// TIA Portal project "V1.3" (V16)

(* hardware
DEVICE "S7-1200 station_1"  S7-1200 Station
   slot 0: "Rack_0"  S7-1200 Rack  Rack  V1.0
   slot 1: "PLC_1"  CPU 1214C DC/DC/DC  6ES7 214-1AG40-0XB0  V4.2
   slot 2: "DI 16/DQ 16x24VDC_1"  6ES7 223-1BL32-0XB0  V2.0
   slot 3: "DI 16x24VDC/DQ 16xRelay_1"  SM 1223 DI16/DQ16 x relay  6ES7 223-1PL32-0XB0  V2.0
   slot 3: "AI 1x12BIT_1"  AI1 signal board  6ES7 231-4HA30-0XB0  V2.0
DEVICE "HMI_1"  KTP700 Basic PN
   slot 0: "HMI_1"  KTP700 Basic PN  6AV2 123-2GB03-0AX0  15.0.0.0
   slot 1: "HMI_RT_1"  KTP700 Basic PN  6AV2 123-2GB03-0AX0  15.0.0.0
   slot 5: "HMI_1.IE_CP_1"  PROFINET Interface  15.0.0.0
      slot 1: "PROFINET Interface_1"  PROFINET Interface
         slot 1: "Port_1"  Port
*)

// ===== PLC "PLC_1"  CPU 1214C DC/DC/DC =====

VAR_GLOBAL   // PLC tag table "Default tag table"
   "czujnik ciśnienia powietrza" AT %I0.0 : Bool;
   "ESTOP" AT %I0.1 : Bool;
   "[P] załączenie powietrza" AT %I0.2 : Bool;
   "[P] wyłączenie powietrza [NC]" AT %I0.3 : Bool;
   "[P] załączenie pompy hydraulicznej" AT %I0.4 : Bool;
   "[P] wyłączenie pompy hydraulicznej [NC]" AT %I0.5 : Bool;
   "[P] przycisk dwuręczny [NC]" AT %I0.6 : Bool;
   "[P] przycisk dwuręczny [NO]" AT %I0.7 : Bool;
   "SQ1" AT %I1.0 : Bool;
   "SQ2" AT %I1.1 : Bool;
   "SQ3" AT %I1.2 : Bool;
   "SQ4" AT %I1.3 : Bool;
   "SQ5" AT %I1.4 : Bool;
   "SQ6" AT %I1.5 : Bool;
   "Bit_1" AT %I8.0 : Bool;
   "Bit_2" AT %I8.1 : Bool;
   "Bit_3" AT %I8.2 : Bool;
   "Bit_4" AT %I8.3 : Bool;
   "Bit_5" AT %I8.4 : Bool;
   "Bit_6" AT %I8.5 : Bool;
   "zwierny_1" AT %I8.6 : Bool;
   "zwierny_2" AT %I8.7 : Bool;
   "zwierny_3" AT %I9.0 : Bool;
   "zwierny_4" AT %I9.1 : Bool;
   "zwierny_5" AT %I9.2 : Bool;
   "zwierny_6" AT %I9.3 : Bool;
   "-" AT %I9.4 : Bool;
   "-(1)" AT %I9.5 : Bool;
   "-(2)" AT %I9.6 : Bool;
   "-(3)" AT %I9.7 : Bool;
   "-(4)" AT %I12.0 : Bool;
   "-(5)" AT %I12.1 : Bool;
   "-(6)" AT %I12.2 : Bool;
   "-(7)" AT %I12.3 : Bool;
   "-(8)" AT %I12.4 : Bool;
   "-(9)" AT %I12.5 : Bool;
   "-(10)" AT %I12.6 : Bool;
   "Kurtyna" AT %I12.7 : Bool;
   "-(12)" AT %I13.0 : Bool;
   "-(13)" AT %I13.1 : Bool;
   "-(14)" AT %I13.2 : Bool;
   "-(15)" AT %I13.3 : Bool;
   "-(16)" AT %I13.4 : Bool;
   "-(17)" AT %I13.5 : Bool;
   "-(18)" AT %I13.6 : Bool;
   "-(19)" AT %I13.7 : Bool;
   "Ciśnienie oleju hydraulicznego" AT %IW80 : Int;
   "Z.H 0" AT %Q0.0 : Bool;
   "Z.H 1" AT %Q0.1 : Bool;
   "Z.H 2" AT %Q0.2 : Bool;
   "Z.H 3" AT %Q0.3 : Bool;
   "Z.H 4" AT %Q0.4 : Bool;
   "Z.H 5" AT %Q0.5 : Bool;
   "Z.H 6" AT %Q0.6 : Bool;
   "Z.H 7" AT %Q0.7 : Bool;
   "Z.H 8" AT %Q1.0 : Bool;
   "-(20)" AT %Q1.1 : Bool;
   "[L] Zawór główny powietrza" AT %Q8.0 : Bool;
   "[L] Pompa hydrauliczna" AT %Q8.1 : Bool;
   "-(21)" AT %Q8.2 : Bool;
   "-(22)" AT %Q8.3 : Bool;
   "-(23)" AT %Q8.4 : Bool;
   "-(24)" AT %Q8.5 : Bool;
   "-(25)" AT %Q8.6 : Bool;
   "-(26)" AT %Q8.7 : Bool;
   "Proces1" AT %Q9.0 : Bool;
   "Proces2" AT %Q9.1 : Bool;
   "Proces3" AT %Q9.2 : Bool;
   "Proces4" AT %Q9.3 : Bool;
   "Proces5" AT %Q9.4 : Bool;
   "Proces6" AT %Q9.5 : Bool;
   "Proces7" AT %Q9.6 : Bool;
   "Proces8" AT %Q9.7 : Bool;
   "Z.P 0" AT %Q12.0 : Bool;
   "Z.P 1" AT %Q12.1 : Bool;
   "Z.P 2" AT %Q12.2 : Bool;
   "Z.P 3" AT %Q12.3 : Bool;
   "Z.P 4" AT %Q12.4 : Bool;
   "smar 1" AT %Q12.5 : Bool;
   "smar 2" AT %Q12.6 : Bool;
   "-(27)" AT %Q12.7 : Bool;
   "-(28)" AT %Q13.0 : Bool;
   "-(29)" AT %Q13.1 : Bool;
   "-(30)" AT %Q13.2 : Bool;
   "-(31)" AT %Q13.3 : Bool;
   "Pompa hydrauliczna" AT %Q13.4 : Bool;
   "-(33)" AT %Q13.5 : Bool;
   "-(34)" AT %Q13.6 : Bool;
   "-(35)" AT %Q13.7 : Bool;
   "Bit1(1)" AT %M0.0 : Bool;
   "Bit2(1)" AT %M0.1 : Bool;
   "Bit3(1)" AT %M0.2 : Bool;
   "Bit4(1)" AT %M0.3 : Bool;
   "Bit5(1)" AT %M0.4 : Bool;
   "Bit6(1)" AT %M0.5 : Bool;
   "Byte0" AT %MB0 : Byte;
   "Tag_1" AT %M7000.0 : Bool;
   "Tag_2" AT %M7000.1 : Bool;
   "Tag_3" AT %M7000.2 : Bool;
   "Tag_4" AT %M7000.5 : Bool;
END_VAR

DATA_BLOCK "main_DB"   // DB2
{ S7_Optimized_Access := 'TRUE' }
VERSION : 0.1
   VAR
      "M" : Array[0..254] of Bool;
      Button : Struct
         Screen_0 : Struct
            Reset_counter_1 : Bool;
            Reset_counter_2 : Bool;
            Lubrication_test : Bool;
            Lubrication_test_1 : Bool;
            Lubrication_test_2 : Bool;
         END_STRUCT;
         Screen_2 : Struct
            "Z.P 0" : Bool;
            "Z.P 1" : Bool;
            "Z.P 2" : Bool;
            "Z.P 3" : Bool;
            "Z.P 4" : Bool;
            "Z.H 0" : Bool;
            "Z.H 1" : Bool;
            "Z.H 2" : Bool;
            "Z.H 3" : Bool;
            "Z.H 4" : Bool;
            "Z.H 5" : Bool;
            "Z.H 6" : Bool;
            "Z.H 7" : Bool;
            "Z.H 8" : Bool;
            Manual_control : Bool;
            Hydraulic_Pump : Bool;
            Relaxation : Bool;
         END_STRUCT;
         Screen_1 : Struct
            "0" : Bool;
         END_STRUCT;
         Screen_3 : Struct
            "0" : Bool;
         END_STRUCT;
         Template : Struct
            "Browsed_punch_+" : Bool;
            "Browsed_punch_-" : Bool;
         END_STRUCT;
      END_STRUCT;
      Status : Struct
         Blink : Bool;
         Manual_control : Bool;
         Browsing_punch : Bool;
         "Two-handed_button" : Bool;
         relaxation : Bool;
         Cycle_time_overload : Bool;
         Lubrication1 : Bool;
         Lubrication2 : Bool;
      END_STRUCT;
   END_VAR
   VAR RETAIN
      var : Struct
         Browsed_punch : Byte;
         Connected_punch : Byte;
         Result_punch : Byte;
         Hydraulic_oil_pressure : Real;
         Lubrication_dur : Time;
         Lubrication_frequency : Int := 1;
         "Descryption Z.P 1" : String;
         "Descryption Z.P 2" : String;
         "Descryption Z.P 3" : String;
         "Descryption Z.P 4" : String;
         "Descryption Z.H 1" : String;
         "Descryption Z.H 2" : String;
         "Descryption Z.H 3" : String;
         "Descryption Z.H 4" : String;
         "Descryption Z.H 5" : String;
         "Descryption Z.H 6" : String;
         "Descryption Z.H 7" : String;
         "Descryption Z.H 8" : String;
         "Descryption SQ 1" : String;
         "Descryption SQ 2" : String;
         "Descryption SQ 3" : String;
         "Descryption SQ 4" : String;
         "Descryption SQ 5" : String;
         "Descryption SQ 6" : String;
         "Descryption contact_sensor 1" : String;
         "Descryption contact_sensor 2" : String;
         "Descryption contact_sensor 3" : String;
         "Descryption contact_sensor 4" : String;
         "Descryption contact_sensor 5" : String;
         "Descryption contact_sensor 6" : String;
      END_STRUCT;
   END_VAR
   VAR
      Timers : Struct
         "0" : IEC_TIMER;
         "1" : IEC_TIMER;
         "2" : IEC_TIMER;
         "3" : IEC_TIMER;
         "4" : IEC_TIMER;
         "5" : IEC_TIMER;
         "6" : IEC_TIMER;
         "7" : IEC_TIMER;
         "8" : IEC_TIMER;
         "9" : IEC_TIMER;
         "10" : IEC_TIMER;
         "11" : IEC_TIMER;
         "12" : IEC_TIMER;
         "13" : IEC_TIMER;
         "14" : IEC_TIMER;
         "15" : IEC_TIMER;
         "16" : IEC_TIMER;
         "17" : IEC_TIMER;
         "18" : IEC_TIMER;
         "19" : IEC_TIMER;
         "20" : IEC_TIMER;
         "21" : IEC_TIMER;
         "22" : IEC_TIMER;
         "23" : IEC_TIMER;
         "24" : IEC_TIMER;
      END_STRUCT;
   END_VAR
BEGIN
END_DATA_BLOCK

DATA_BLOCK "Counters"   // DB5
{ S7_Optimized_Access := 'TRUE' }
VERSION : 0.1
   VAR RETAIN
      Counter_1 : Int;
      Counter_2 : Int;
   END_VAR
   VAR
      Lubricatons : Int := 1;
   END_VAR
BEGIN
END_DATA_BLOCK

DATA_BLOCK "Punch_parameters"   // DB6
{ S7_Optimized_Access := 'TRUE' }
VERSION : 0.1
   VAR
      Punch : Array[0..10] of Struct
         "Z.P 1" : String;
         "Z.P 2" : String;
         "Z.P 3" : String;
         "Z.P 4" : String;
         "Z.H 1" : String;
         "Z.H 2" : String;
         "Z.H 3" : String;
         "Z.H 4" : String;
         "Z.H 5" : String;
         "Z.H 6" : String;
         "Z.H 7" : String;
         "Z.H 8" : String;
         SQ1 : String;
         SQ2 : String;
         SQ3 : String;
         SQ4 : String;
         SQ5 : String;
         SQ6 : String;
         Contact_sensor_1 : String;
         Contact_sensor_2 : String;
         Contact_sensor_3 : String;
         Contact_sensor_4 : String;
         Contact_sensor_5 : String;
         Contact_sensor_6 : String;
      END_STRUCT;
   END_VAR
BEGIN
   Punch[1]."Z.H 5" := 'Lewy naprzod';
   Punch[1]."Z.H 6" := 'Lewy wstecz';
   Punch[1]."Z.H 7" := 'Prawy naprzod';
   Punch[1]."Z.H 8" := 'Prawy wstecz';
   Punch[1].SQ1 := 'Lewy z tylu [NC]';
   Punch[1].SQ2 := 'Lewy z przodu';
   Punch[1].SQ3 := 'Prawy z tylu';
   Punch[1].SQ4 := 'Prawy z przodu';
   Punch[1].Contact_sensor_1 := 'Przy lewym silowniku';
   Punch[1].Contact_sensor_2 := 'Przy prawym silowniku 1';
   Punch[1].Contact_sensor_3 := 'Przy prawym silowniku 2';
   Punch[1]."Z.P 1" := 'Klamra';
   Punch[1]."Z.P 2" := 'Baza';
   Punch[1].SQ5 := 'Klamra zacisnieta';
   Punch[2]."Z.P 1" := 'Baza';
   Punch[2]."Z.P 2" := 'Kon';
   Punch[2].SQ3 := 'Kon';
   Punch[2]."Z.H 1" := 'Silownik naprzod';
   Punch[2]."Z.H 2" := 'Silownik wstecz';
   Punch[2].SQ1 := 'Silownik przod';
   Punch[2].SQ2 := 'Silownik tyl';
   Punch[2].Contact_sensor_1 := '1';
   Punch[2].Contact_sensor_2 := '2';
   Punch[3]."Z.P 1" := 'Kon 1';
   Punch[3]."Z.P 2" := 'Kon 2';
   Punch[3]."Z.H 3" := 'Silownik naprzod';
   Punch[3]."Z.H 4" := 'Silownik wstecz';
   Punch[3].SQ1 := 'Silownik przod';
   Punch[3].SQ2 := 'Silownik tyl';
   Punch[3].SQ3 := 'Kon 1';
   Punch[3].SQ4 := 'Kon 2';
   Punch[3].Contact_sensor_1 := '1';
   Punch[3].Contact_sensor_2 := '2';
   Punch[4].SQ1 := 'Prawy stempel wysuniety';
   Punch[4].Contact_sensor_1 := '1';
   Punch[4].SQ2 := 'Prawy stempel wycofany';
   Punch[4].SQ3 := 'Lewy stempel wysuniety';
   Punch[4].SQ4 := 'Lewy stempel wycofany';
   Punch[4]."Z.H 1" := 'L st. wysuniecie';
   Punch[4]."Z.H 2" := 'L st. wycofanie';
   Punch[4]."Z.H 3" := 'P st. wysuniecie';
   Punch[4]."Z.H 4" := 'P st. wycofanie';
   Punch[5]."Z.H 7" := 'Stempel naprzod';
   Punch[5]."Z.H 8" := 'Stempel wstecz';
   Punch[5].SQ1 := 'Material dosuniety';
   Punch[5].SQ2 := 'Stempel wycofany';
END_DATA_BLOCK

DATA_BLOCK "Relaxation_DB"   // DB7
{ S7_Optimized_Access := 'TRUE' }
VERSION : 0.1
// stored: InstanceOfName Relaxation
"Relaxation"
BEGIN
END_DATA_BLOCK

// folder: Punch_blocks

DATA_BLOCK "Punch1_DB"   // DB1
{ S7_Optimized_Access := 'TRUE' }
VERSION : 0.1
// stored: InstanceOfName Punch1
"Punch1"
BEGIN
END_DATA_BLOCK

DATA_BLOCK "Punch2_DB"   // DB3
{ S7_Optimized_Access := 'TRUE' }
VERSION : 0.1
// stored: InstanceOfName Punch2
"Punch2"
BEGIN
END_DATA_BLOCK

DATA_BLOCK "Punch3_DB"   // DB4
{ S7_Optimized_Access := 'TRUE' }
VERSION : 0.1
// stored: InstanceOfName Punch3
"Punch3"
BEGIN
END_DATA_BLOCK

DATA_BLOCK "Punch4_DB"   // DB15
{ S7_Optimized_Access := 'TRUE' }
VERSION : 0.1
// stored: InstanceOfName Punch4
"Punch4"
BEGIN
END_DATA_BLOCK

DATA_BLOCK "Punch5_DB"   // DB16
{ S7_Optimized_Access := 'TRUE' }
VERSION : 0.1
// stored: InstanceOfName Punch5
"Punch5"
BEGIN
END_DATA_BLOCK

// folder: System blocks/Program resources

DATA_BLOCK "IEC_Timer_0_DB"   // DB8
{ S7_Optimized_Access := 'TRUE' }
AUTHOR : Simatic
FAMILY : IEC
NAME : IEC_TMR
VERSION : 1.0
// stored: InstanceOfName IEC_TIMER
"IEC_TIMER"
BEGIN
END_DATA_BLOCK

DATA_BLOCK "IEC_Timer_0_DB_1"   // DB9
{ S7_Optimized_Access := 'TRUE' }
AUTHOR : Simatic
FAMILY : IEC
NAME : IEC_TMR
VERSION : 1.0
// stored: InstanceOfName IEC_TIMER
"IEC_TIMER"
BEGIN
END_DATA_BLOCK

DATA_BLOCK "IEC_Timer_0_DB_2"   // DB10
{ S7_Optimized_Access := 'TRUE' }
AUTHOR : Simatic
FAMILY : IEC
NAME : IEC_TMR
VERSION : 1.0
// stored: InstanceOfName IEC_TIMER
"IEC_TIMER"
BEGIN
END_DATA_BLOCK

DATA_BLOCK "IEC_Timer_0_DB_3"   // DB11
{ S7_Optimized_Access := 'TRUE' }
AUTHOR : Simatic
FAMILY : IEC
NAME : IEC_TMR
VERSION : 1.0
// stored: InstanceOfName IEC_TIMER
"IEC_TIMER"
BEGIN
END_DATA_BLOCK

DATA_BLOCK "IEC_Timer_0_DB_4"   // DB12
{ S7_Optimized_Access := 'TRUE' }
AUTHOR : Simatic
FAMILY : IEC
NAME : IEC_TMR
VERSION : 1.0
// stored: InstanceOfName IEC_TIMER
"IEC_TIMER"
BEGIN
END_DATA_BLOCK

DATA_BLOCK "IEC_Timer_0_DB_5"   // DB13
{ S7_Optimized_Access := 'TRUE' }
AUTHOR : Simatic
FAMILY : IEC
NAME : IEC_TMR
VERSION : 1.0
// stored: InstanceOfName IEC_TIMER
"IEC_TIMER"
BEGIN
END_DATA_BLOCK

DATA_BLOCK "IEC_Timer_0_DB_6"   // DB14
{ S7_Optimized_Access := 'TRUE' }
AUTHOR : Simatic
FAMILY : IEC
NAME : IEC_TMR
VERSION : 1.0
// stored: InstanceOfName IEC_TIMER
"IEC_TIMER"
BEGIN
END_DATA_BLOCK

// folder: (top level)

FUNCTION_BLOCK "Relaxation"   // FB4, LAD
{ S7_Optimized_Access := 'TRUE' }
VERSION : 0.1
   VAR_INPUT
      Activate : Bool;
   END_VAR
   VAR
      finish : Bool;
   END_VAR
   VAR_TEMP   // added for the SCL form of the ladder/FBD networks
      _w1 : Bool;
   END_VAR
BEGIN

REGION Network 1
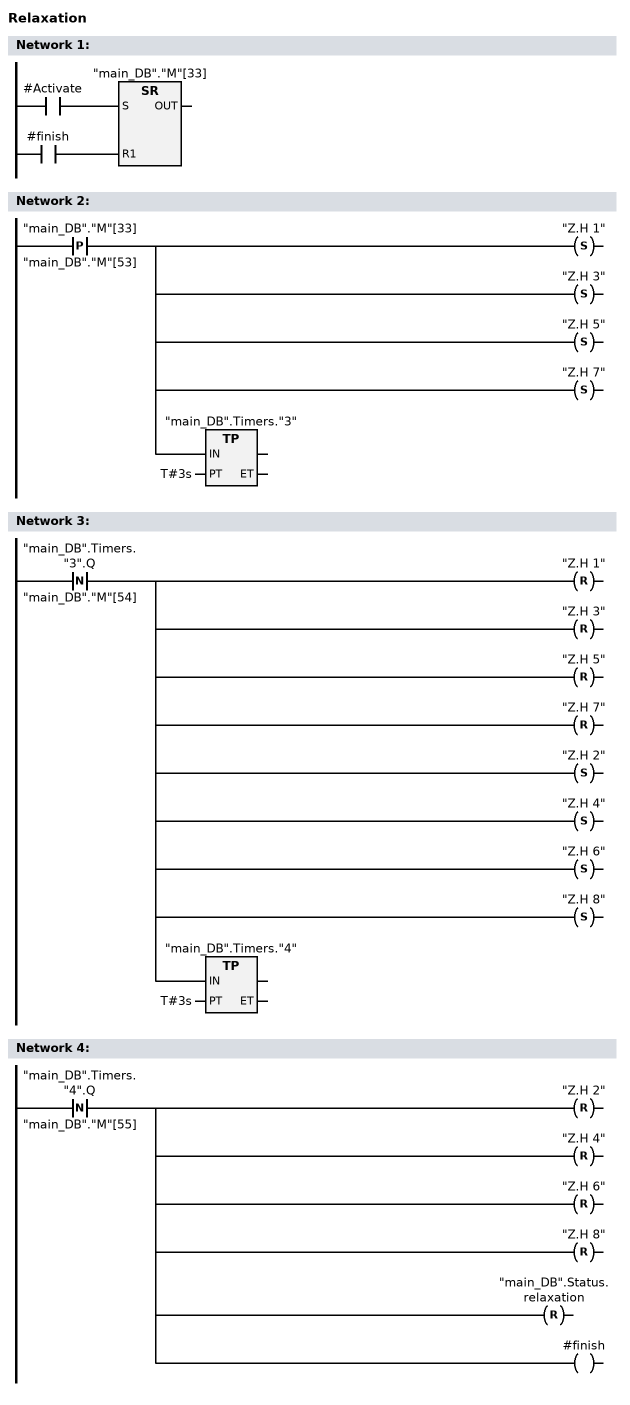
   RUNG wire#powerrail
      Contact( #Activate )
      S_SR(operand := "main_DB"."M"[33], r1 := wire#w1)
   END_RUNG
   RUNG wire#powerrail
      Contact( #finish )
   END_RUNG wire#w1
   // the same network as SCL:
   IF #Activate THEN
       "main_DB"."M"[33] := TRUE;   // SR flip-flop
   END_IF;
   IF #finish THEN "main_DB"."M"[33] := FALSE; END_IF;
END_REGION

REGION Network 2
   #_w1 := "main_DB"."M"[33] AND NOT "main_DB"."M"[53];   // rising edge of "main_DB"."M"[33]
   "main_DB"."M"[53] := "main_DB"."M"[33];
   IF #_w1 THEN
       "Z.H 1" := TRUE;
       "Z.H 3" := TRUE;
       "Z.H 5" := TRUE;
       "Z.H 7" := TRUE;
   END_IF;
   "main_DB".Timers."3".TP(IN := #_w1, PT := T#3s);
END_REGION

REGION Network 3
   #_w1 := NOT "main_DB".Timers."3".Q AND "main_DB"."M"[54];   // falling edge of "main_DB".Timers."3".Q
   "main_DB"."M"[54] := "main_DB".Timers."3".Q;
   IF #_w1 THEN
       "Z.H 1" := FALSE;
       "Z.H 3" := FALSE;
       "Z.H 5" := FALSE;
       "Z.H 7" := FALSE;
       "Z.H 2" := TRUE;
       "Z.H 4" := TRUE;
       "Z.H 6" := TRUE;
       "Z.H 8" := TRUE;
   END_IF;
   "main_DB".Timers."4".TP(IN := #_w1, PT := T#3s);
END_REGION

REGION Network 4
   RUNG wire#powerrail
      N_Contact(operand := "main_DB".Timers."4".Q, bit := "main_DB"."M"[55])
      wire#w1
      R_Coil( "Z.H 2" )
   END_RUNG
   RUNG wire#w1
      R_Coil( "Z.H 4" )
   END_RUNG
   RUNG wire#w1
      R_Coil( "Z.H 6" )
   END_RUNG
   RUNG wire#w1
      R_Coil( "Z.H 8" )
   END_RUNG
   RUNG wire#w1
      R_Coil( "main_DB".Status.relaxation )
   END_RUNG
   RUNG wire#w1
      Coil( #finish )
   END_RUNG
   // the same network as SCL:
   #_w1 := NOT "main_DB".Timers."4".Q AND "main_DB"."M"[55];   // falling edge of "main_DB".Timers."4".Q
   "main_DB"."M"[55] := "main_DB".Timers."4".Q;
   IF #_w1 THEN
       "Z.H 2" := FALSE;
       "Z.H 4" := FALSE;
       "Z.H 6" := FALSE;
       "Z.H 8" := FALSE;
       "main_DB".Status.relaxation := FALSE;
   END_IF;
   #finish := #_w1;
END_REGION
END_FUNCTION_BLOCK

FUNCTION "SR_Switch" : Void   // FC1, LAD
{ S7_Optimized_Access := 'TRUE' }
VERSION : 0.1
   VAR_INPUT
      Input : Bool;
   END_VAR
   VAR_IN_OUT
      "M" : Bool;
      M1 : Bool;
      Out : Bool;
   END_VAR
   VAR_TEMP
      N : Bool;
      N1 : Bool;
   END_VAR
   VAR_TEMP   // added for the SCL form of the ladder/FBD networks
      _w1 : Bool;
      _w2 : Bool;
   END_VAR
BEGIN

REGION Network 1
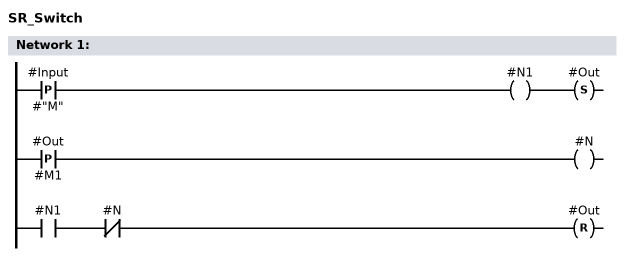
   RUNG wire#powerrail
      P_Contact(operand := #Input, bit := #"M")
      Coil( #N1 )
      S_Coil( #Out )
   END_RUNG
   RUNG wire#powerrail
      P_Contact(operand := #Out, bit := #M1)
      Coil( #N )
   END_RUNG
   RUNG wire#powerrail
      Contact( #N1 )
      I_Contact( #N )
      R_Coil( #Out )
   END_RUNG
   // the same network as SCL:
   #_w1 := #Input AND NOT #"M";   // rising edge of #Input
   #"M" := #Input;
   #N1 := #_w1;
   IF #_w1 THEN #Out := TRUE; END_IF;
   #_w2 := #Out AND NOT #M1;   // rising edge of #Out
   #M1 := #Out;
   #N := #_w2;
   IF #N1 AND NOT #N THEN #Out := FALSE; END_IF;
END_REGION
END_FUNCTION

FUNCTION "Outputs_reset" : Void   // FC2, LAD
{ S7_Optimized_Access := 'TRUE' }
VERSION : 0.1
BEGIN

REGION Network 1
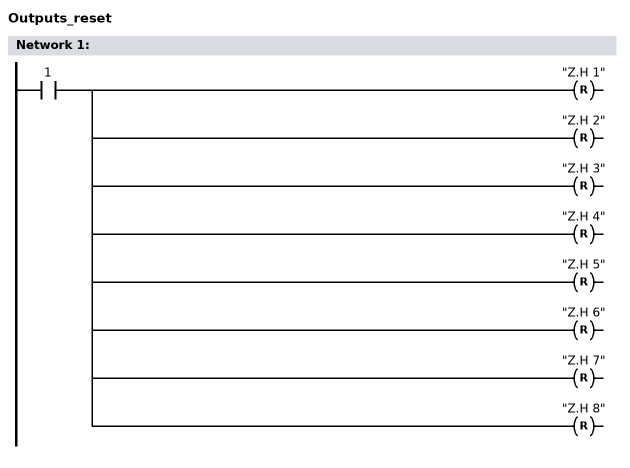
   RUNG wire#powerrail
      Contact( 1 )
      wire#w1
      R_Coil( "Z.H 1" )
   END_RUNG
   RUNG wire#w1
      R_Coil( "Z.H 2" )
   END_RUNG
   RUNG wire#w1
      R_Coil( "Z.H 3" )
   END_RUNG
   RUNG wire#w1
      R_Coil( "Z.H 4" )
   END_RUNG
   RUNG wire#w1
      R_Coil( "Z.H 5" )
   END_RUNG
   RUNG wire#w1
      R_Coil( "Z.H 6" )
   END_RUNG
   RUNG wire#w1
      R_Coil( "Z.H 7" )
   END_RUNG
   RUNG wire#w1
      R_Coil( "Z.H 8" )
   END_RUNG
   // the same network as SCL:
   IF 1 THEN
       "Z.H 1" := FALSE;
       "Z.H 2" := FALSE;
       "Z.H 3" := FALSE;
       "Z.H 4" := FALSE;
       "Z.H 5" := FALSE;
       "Z.H 6" := FALSE;
       "Z.H 7" := FALSE;
       "Z.H 8" := FALSE;
   END_IF;
END_REGION
END_FUNCTION

ORGANIZATION_BLOCK "Main"   // OB1, LAD, ProgramCycle
TITLE = "Main Program Sweep (Cycle)"
{ S7_Optimized_Access := 'TRUE' }
VERSION : 0.1
   VAR_INPUT
      Initial_Call : Bool;   // Initial call of this OB
      Remanence : Bool;   // =True, if remanent data are available
   END_VAR
   VAR_TEMP
      X : Real;
   END_VAR
   VAR_TEMP   // added for the SCL form of the ladder/FBD networks
      _w1 : Bool;
      _w2 : Bool;
      _w3 : Bool;
      _w4 : Bool;
      _w5 : Bool;
      _w6 : Bool;
      _w7 : Bool;
      _w8 : Bool;
      _w9 : Bool;
      _w10 : Bool;
      _w11 : Bool;
      _w12 : Bool;
      _w13 : Bool;
      _w14 : Bool;
      _w15 : Bool;
      _w16 : Bool;
      _w17 : Bool;
      _w18 : Bool;
      _w19 : Bool;
      _w20 : Bool;
      _w21 : Bool;
      _w22 : Bool;
      _w23 : Bool;
      _w24 : Bool;
   END_VAR
BEGIN

REGION Network 1 (SCL): Conversion Connected_punch
   "Bit1(1)" := "Bit_1";
   "Bit2(1)" := "Bit_2";
   "Bit3(1)" := "Bit_3";
   "Bit4(1)" := "Bit_4";
   "Bit5(1)" := "Bit_5";
   "Bit6(1)" := "Bit_6";

   "main_DB".var.Connected_punch := "Byte0";
END_REGION

REGION Network 2 (SCL): Browsed_punch
   IF "main_DB".Button.Template."Browsed_punch_+" AND NOT "main_DB".M[34] THEN
       IF "main_DB".var.Browsed_punch = 63 THEN
           "main_DB".var.Browsed_punch := 0;
           ;
       ELSE
           "main_DB".var.Browsed_punch := "main_DB".var.Browsed_punch + 1;
           ;
       END_IF;
       ;
   END_IF;
   "main_DB".M[34] := "main_DB".Button.Template."Browsed_punch_+";

   IF "main_DB".Button.Template."Browsed_punch_-" AND NOT "main_DB".M[35] THEN
       IF "main_DB".var.Browsed_punch = 0 THEN
           "main_DB".var.Browsed_punch := 63;
           ;
       ELSE
           "main_DB".var.Browsed_punch := "main_DB".var.Browsed_punch - 1;
           ;
       END_IF;

       ;
   END_IF;
   "main_DB".M[35] := "main_DB".Button.Template."Browsed_punch_-";

   IF "main_DB".var.Connected_punch <> 0 THEN
       "main_DB".var.Browsed_punch := 0;
       ;
   END_IF;
END_REGION

REGION Network 3 (SCL): Result_punch
   IF "main_DB".var.Connected_punch = 0 THEN
       "main_DB".var.Result_punch := "main_DB".var.Browsed_punch;
       ;
   ELSE
       "main_DB".var.Result_punch := "main_DB".var.Connected_punch;
       ;
   END_IF;
END_REGION

REGION Network 4: Punch 1
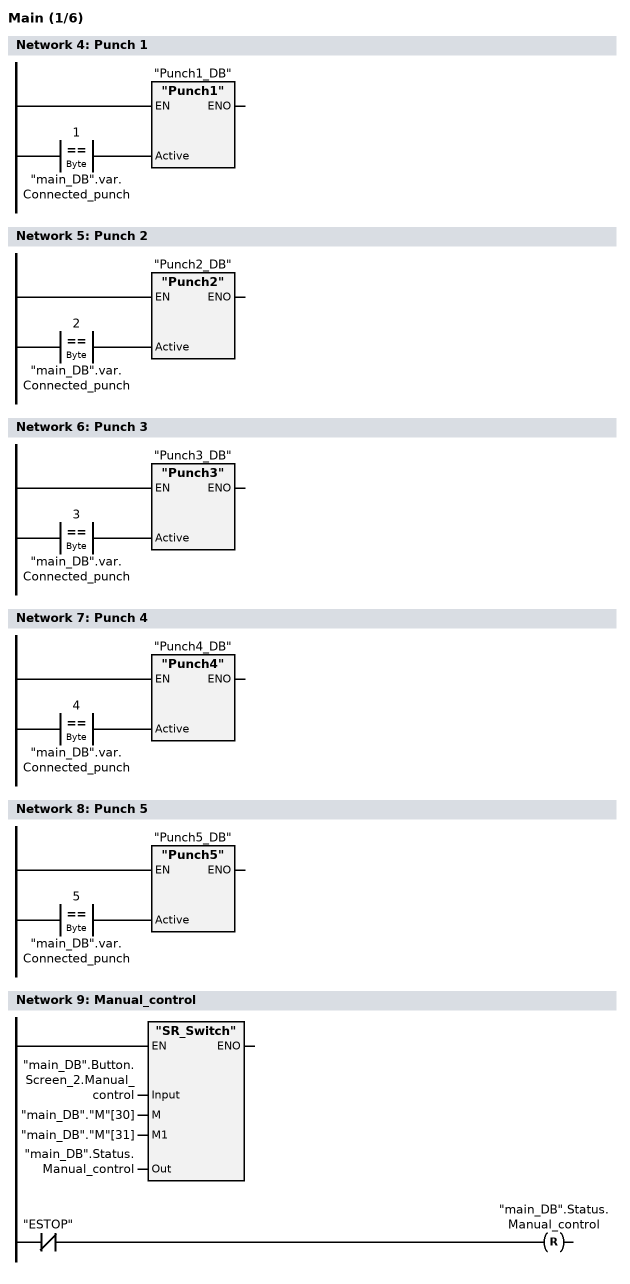
   RUNG wire#powerrail
      "Punch1_DB"(Active := wire#w1)
   END_RUNG
   RUNG wire#powerrail
      { S7_Templates := "SrcType := Byte" } EQ_Contact(in1 := 1, in2 := "main_DB".var.Connected_punch)
   END_RUNG wire#w1
   // the same network as SCL:
   "Punch1_DB"(Active := 1 = "main_DB".var.Connected_punch);   // "Punch1"
END_REGION

REGION Network 5: Punch 2
   RUNG wire#powerrail
      "Punch2_DB"(Active := wire#w1)
   END_RUNG
   RUNG wire#powerrail
      { S7_Templates := "SrcType := Byte" } EQ_Contact(in1 := 2, in2 := "main_DB".var.Connected_punch)
   END_RUNG wire#w1
   // the same network as SCL:
   "Punch2_DB"(Active := 2 = "main_DB".var.Connected_punch);   // "Punch2"
END_REGION

REGION Network 6: Punch 3
   RUNG wire#powerrail
      "Punch3_DB"(Active := wire#w1)
   END_RUNG
   RUNG wire#powerrail
      { S7_Templates := "SrcType := Byte" } EQ_Contact(in1 := 3, in2 := "main_DB".var.Connected_punch)
   END_RUNG wire#w1
   // the same network as SCL:
   "Punch3_DB"(Active := 3 = "main_DB".var.Connected_punch);   // "Punch3"
END_REGION

REGION Network 7: Punch 4
   RUNG wire#powerrail
      "Punch4_DB"(Active := wire#w1)
   END_RUNG
   RUNG wire#powerrail
      { S7_Templates := "SrcType := Byte" } EQ_Contact(in1 := 4, in2 := "main_DB".var.Connected_punch)
   END_RUNG wire#w1
   // the same network as SCL:
   "Punch4_DB"(Active := 4 = "main_DB".var.Connected_punch);   // "Punch4"
END_REGION

REGION Network 8: Punch 5
   RUNG wire#powerrail
      "Punch5_DB"(Active := wire#w1)
   END_RUNG
   RUNG wire#powerrail
      { S7_Templates := "SrcType := Byte" } EQ_Contact(in1 := 5, in2 := "main_DB".var.Connected_punch)
   END_RUNG wire#w1
   // the same network as SCL:
   "Punch5_DB"(Active := 5 = "main_DB".var.Connected_punch);   // "Punch5"
END_REGION

REGION Network 9: Manual_control
   RUNG wire#powerrail
      "SR_Switch"(Input := "main_DB".Button.Screen_2.Manual_control, "M" := "main_DB"."M"[30], M1 := "main_DB"."M"[31], Out := "main_DB".Status.Manual_control)
   END_RUNG
   RUNG wire#powerrail
      I_Contact( "ESTOP" )
      R_Coil( "main_DB".Status.Manual_control )
   END_RUNG
   // the same network as SCL:
   "SR_Switch"(Input := "main_DB".Button.Screen_2.Manual_control,
               "M" := "main_DB"."M"[30],
               M1 := "main_DB"."M"[31],
               Out := "main_DB".Status.Manual_control);
   IF NOT "ESTOP" THEN "main_DB".Status.Manual_control := FALSE; END_IF;
END_REGION

REGION Network 10: Manual pneumatics
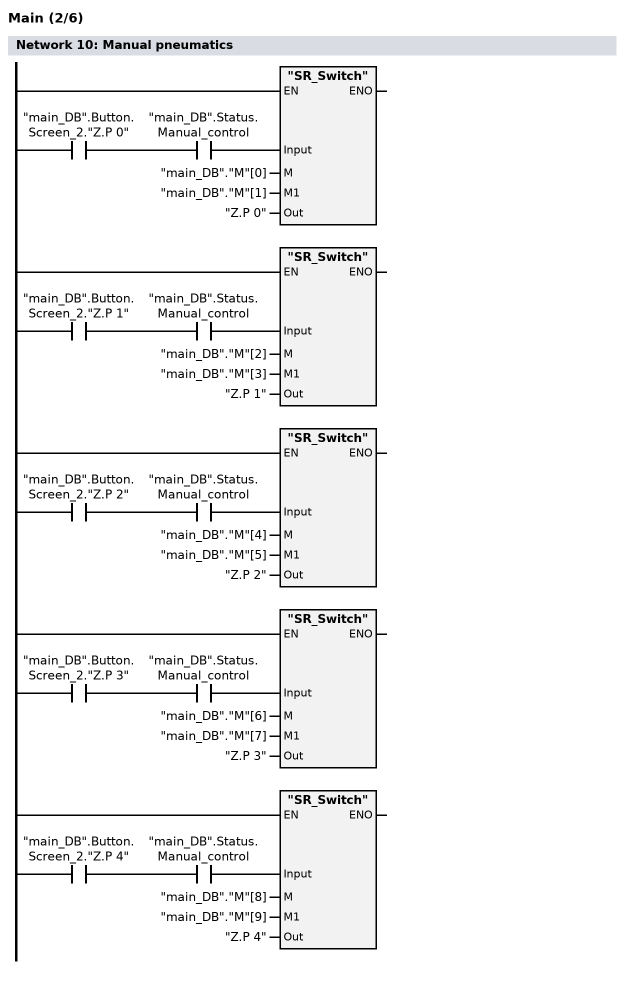
   RUNG wire#powerrail
      "SR_Switch"(Input := wire#w1, "M" := "main_DB"."M"[0], M1 := "main_DB"."M"[1], Out := "Z.P 0")
   END_RUNG
   RUNG wire#powerrail
      Contact( "main_DB".Button.Screen_2."Z.P 0" )
      Contact( "main_DB".Status.Manual_control )
   END_RUNG wire#w1
   RUNG wire#powerrail
      "SR_Switch"(Input := wire#w2, "M" := "main_DB"."M"[2], M1 := "main_DB"."M"[3], Out := "Z.P 1")
   END_RUNG
   RUNG wire#powerrail
      Contact( "main_DB".Button.Screen_2."Z.P 1" )
      Contact( "main_DB".Status.Manual_control )
   END_RUNG wire#w2
   RUNG wire#powerrail
      "SR_Switch"(Input := wire#w3, "M" := "main_DB"."M"[4], M1 := "main_DB"."M"[5], Out := "Z.P 2")
   END_RUNG
   RUNG wire#powerrail
      Contact( "main_DB".Button.Screen_2."Z.P 2" )
      Contact( "main_DB".Status.Manual_control )
   END_RUNG wire#w3
   RUNG wire#powerrail
      "SR_Switch"(Input := wire#w4, "M" := "main_DB"."M"[6], M1 := "main_DB"."M"[7], Out := "Z.P 3")
   END_RUNG
   RUNG wire#powerrail
      Contact( "main_DB".Button.Screen_2."Z.P 3" )
      Contact( "main_DB".Status.Manual_control )
   END_RUNG wire#w4
   RUNG wire#powerrail
      "SR_Switch"(Input := wire#w5, "M" := "main_DB"."M"[8], M1 := "main_DB"."M"[9], Out := "Z.P 4")
   END_RUNG
   RUNG wire#powerrail
      Contact( "main_DB".Button.Screen_2."Z.P 4" )
      Contact( "main_DB".Status.Manual_control )
   END_RUNG wire#w5
   // the same network as SCL:
   "SR_Switch"(Input := "main_DB".Button.Screen_2."Z.P 0" AND "main_DB".Status.Manual_control,
               "M" := "main_DB"."M"[0],
               M1 := "main_DB"."M"[1],
               Out := "Z.P 0");
   "SR_Switch"(Input := "main_DB".Button.Screen_2."Z.P 1" AND "main_DB".Status.Manual_control,
               "M" := "main_DB"."M"[2],
               M1 := "main_DB"."M"[3],
               Out := "Z.P 1");
   "SR_Switch"(Input := "main_DB".Button.Screen_2."Z.P 2" AND "main_DB".Status.Manual_control,
               "M" := "main_DB"."M"[4],
               M1 := "main_DB"."M"[5],
               Out := "Z.P 2");
   "SR_Switch"(Input := "main_DB".Button.Screen_2."Z.P 3" AND "main_DB".Status.Manual_control,
               "M" := "main_DB"."M"[6],
               M1 := "main_DB"."M"[7],
               Out := "Z.P 3");
   "SR_Switch"(Input := "main_DB".Button.Screen_2."Z.P 4" AND "main_DB".Status.Manual_control,
               "M" := "main_DB"."M"[8],
               M1 := "main_DB"."M"[9],
               Out := "Z.P 4");
END_REGION

REGION Network 11: Manual hydraulics
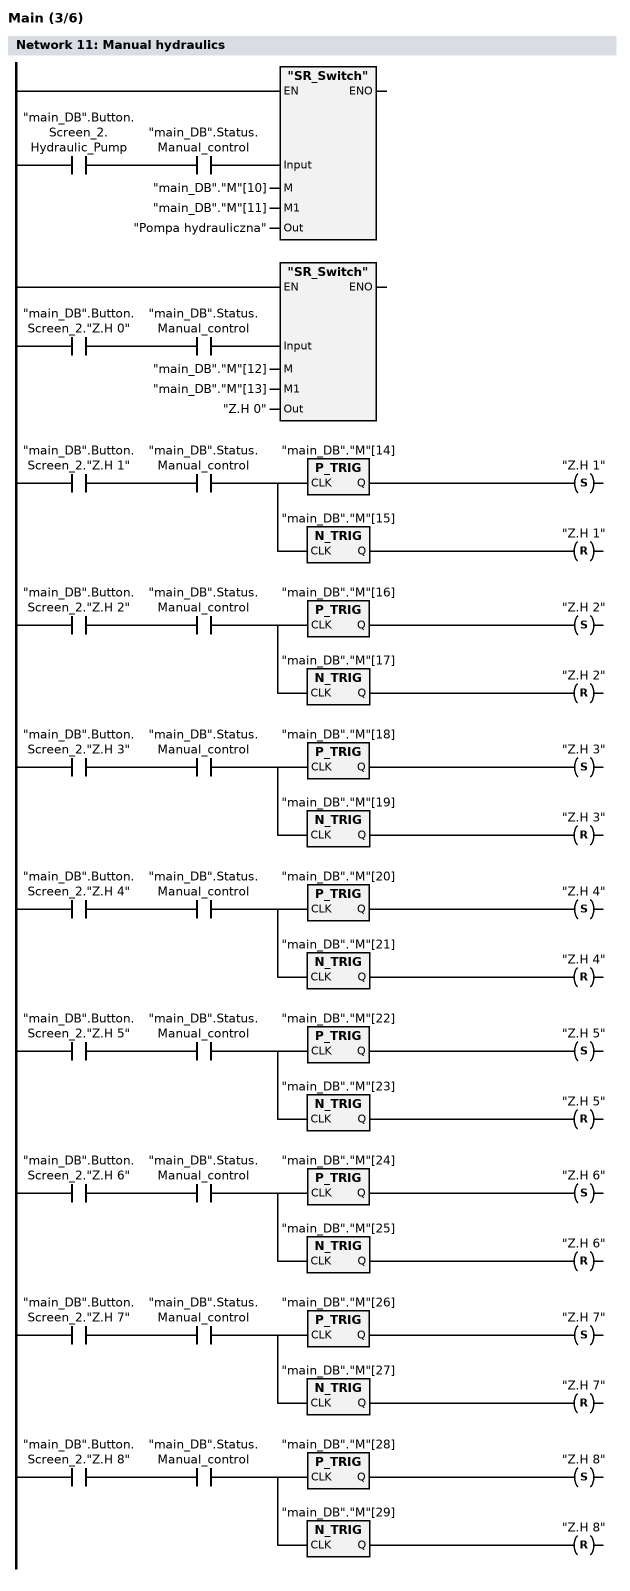
   RUNG wire#powerrail
      "SR_Switch"(Input := wire#w1, "M" := "main_DB"."M"[10], M1 := "main_DB"."M"[11], Out := "Pompa hydrauliczna")
   END_RUNG
   RUNG wire#powerrail
      Contact( "main_DB".Button.Screen_2.Hydraulic_Pump )
      Contact( "main_DB".Status.Manual_control )
   END_RUNG wire#w1
   RUNG wire#powerrail
      "SR_Switch"(Input := wire#w2, "M" := "main_DB"."M"[12], M1 := "main_DB"."M"[13], Out := "Z.H 0")
   END_RUNG
   RUNG wire#powerrail
      Contact( "main_DB".Button.Screen_2."Z.H 0" )
      Contact( "main_DB".Status.Manual_control )
   END_RUNG wire#w2
   RUNG wire#powerrail
      Contact( "main_DB".Button.Screen_2."Z.H 1" )
      Contact( "main_DB".Status.Manual_control )
      wire#w3
      P_Trig( "main_DB"."M"[14] )
      S_Coil( "Z.H 1" )
   END_RUNG
   RUNG wire#w3
      N_Trig( "main_DB"."M"[15] )
      R_Coil( "Z.H 1" )
   END_RUNG
   RUNG wire#powerrail
      Contact( "main_DB".Button.Screen_2."Z.H 2" )
      Contact( "main_DB".Status.Manual_control )
      wire#w4
      P_Trig( "main_DB"."M"[16] )
      S_Coil( "Z.H 2" )
   END_RUNG
   RUNG wire#w4
      N_Trig( "main_DB"."M"[17] )
      R_Coil( "Z.H 2" )
   END_RUNG
   RUNG wire#powerrail
      Contact( "main_DB".Button.Screen_2."Z.H 3" )
      Contact( "main_DB".Status.Manual_control )
      wire#w5
      P_Trig( "main_DB"."M"[18] )
      S_Coil( "Z.H 3" )
   END_RUNG
   RUNG wire#w5
      N_Trig( "main_DB"."M"[19] )
      R_Coil( "Z.H 3" )
   END_RUNG
   RUNG wire#powerrail
      Contact( "main_DB".Button.Screen_2."Z.H 4" )
      Contact( "main_DB".Status.Manual_control )
      wire#w6
      P_Trig( "main_DB"."M"[20] )
      S_Coil( "Z.H 4" )
   END_RUNG
   RUNG wire#w6
      N_Trig( "main_DB"."M"[21] )
      R_Coil( "Z.H 4" )
   END_RUNG
   RUNG wire#powerrail
      Contact( "main_DB".Button.Screen_2."Z.H 5" )
      Contact( "main_DB".Status.Manual_control )
      wire#w7
      P_Trig( "main_DB"."M"[22] )
      S_Coil( "Z.H 5" )
   END_RUNG
   RUNG wire#w7
      N_Trig( "main_DB"."M"[23] )
      R_Coil( "Z.H 5" )
   END_RUNG
   RUNG wire#powerrail
      Contact( "main_DB".Button.Screen_2."Z.H 6" )
      Contact( "main_DB".Status.Manual_control )
      wire#w8
      P_Trig( "main_DB"."M"[24] )
      S_Coil( "Z.H 6" )
   END_RUNG
   RUNG wire#w8
      N_Trig( "main_DB"."M"[25] )
      R_Coil( "Z.H 6" )
   END_RUNG
   RUNG wire#powerrail
      Contact( "main_DB".Button.Screen_2."Z.H 7" )
      Contact( "main_DB".Status.Manual_control )
      wire#w9
      P_Trig( "main_DB"."M"[26] )
      S_Coil( "Z.H 7" )
   END_RUNG
   RUNG wire#w9
      N_Trig( "main_DB"."M"[27] )
      R_Coil( "Z.H 7" )
   END_RUNG
   RUNG wire#powerrail
      Contact( "main_DB".Button.Screen_2."Z.H 8" )
      Contact( "main_DB".Status.Manual_control )
      wire#w10
      P_Trig( "main_DB"."M"[28] )
      S_Coil( "Z.H 8" )
   END_RUNG
   RUNG wire#w10
      N_Trig( "main_DB"."M"[29] )
      R_Coil( "Z.H 8" )
   END_RUNG
   // the same network as SCL:
   "SR_Switch"(Input := "main_DB".Button.Screen_2.Hydraulic_Pump AND "main_DB".Status.Manual_control,
               "M" := "main_DB"."M"[10],
               M1 := "main_DB"."M"[11],
               Out := "Pompa hydrauliczna");
   "SR_Switch"(Input := "main_DB".Button.Screen_2."Z.H 0" AND "main_DB".Status.Manual_control,
               "M" := "main_DB"."M"[12],
               M1 := "main_DB"."M"[13],
               Out := "Z.H 0");
   #_w1 := "main_DB".Button.Screen_2."Z.H 1" AND "main_DB".Status.Manual_control;
   #_w2 := #_w1 AND NOT "main_DB"."M"[14];   // rising edge
   "main_DB"."M"[14] := #_w1;
   IF #_w2 THEN "Z.H 1" := TRUE; END_IF;
   #_w3 := NOT #_w1 AND "main_DB"."M"[15];   // falling edge
   "main_DB"."M"[15] := #_w1;
   IF #_w3 THEN "Z.H 1" := FALSE; END_IF;
   #_w4 := "main_DB".Button.Screen_2."Z.H 2" AND "main_DB".Status.Manual_control;
   #_w5 := #_w4 AND NOT "main_DB"."M"[16];   // rising edge
   "main_DB"."M"[16] := #_w4;
   IF #_w5 THEN "Z.H 2" := TRUE; END_IF;
   #_w6 := NOT #_w4 AND "main_DB"."M"[17];   // falling edge
   "main_DB"."M"[17] := #_w4;
   IF #_w6 THEN "Z.H 2" := FALSE; END_IF;
   #_w7 := "main_DB".Button.Screen_2."Z.H 3" AND "main_DB".Status.Manual_control;
   #_w8 := #_w7 AND NOT "main_DB"."M"[18];   // rising edge
   "main_DB"."M"[18] := #_w7;
   IF #_w8 THEN "Z.H 3" := TRUE; END_IF;
   #_w9 := NOT #_w7 AND "main_DB"."M"[19];   // falling edge
   "main_DB"."M"[19] := #_w7;
   IF #_w9 THEN "Z.H 3" := FALSE; END_IF;
   #_w10 := "main_DB".Button.Screen_2."Z.H 4" AND "main_DB".Status.Manual_control;
   #_w11 := #_w10 AND NOT "main_DB"."M"[20];   // rising edge
   "main_DB"."M"[20] := #_w10;
   IF #_w11 THEN "Z.H 4" := TRUE; END_IF;
   #_w12 := NOT #_w10 AND "main_DB"."M"[21];   // falling edge
   "main_DB"."M"[21] := #_w10;
   IF #_w12 THEN "Z.H 4" := FALSE; END_IF;
   #_w13 := "main_DB".Button.Screen_2."Z.H 5" AND "main_DB".Status.Manual_control;
   #_w14 := #_w13 AND NOT "main_DB"."M"[22];   // rising edge
   "main_DB"."M"[22] := #_w13;
   IF #_w14 THEN "Z.H 5" := TRUE; END_IF;
   #_w15 := NOT #_w13 AND "main_DB"."M"[23];   // falling edge
   "main_DB"."M"[23] := #_w13;
   IF #_w15 THEN "Z.H 5" := FALSE; END_IF;
   #_w16 := "main_DB".Button.Screen_2."Z.H 6" AND "main_DB".Status.Manual_control;
   #_w17 := #_w16 AND NOT "main_DB"."M"[24];   // rising edge
   "main_DB"."M"[24] := #_w16;
   IF #_w17 THEN "Z.H 6" := TRUE; END_IF;
   #_w18 := NOT #_w16 AND "main_DB"."M"[25];   // falling edge
   "main_DB"."M"[25] := #_w16;
   IF #_w18 THEN "Z.H 6" := FALSE; END_IF;
   #_w19 := "main_DB".Button.Screen_2."Z.H 7" AND "main_DB".Status.Manual_control;
   #_w20 := #_w19 AND NOT "main_DB"."M"[26];   // rising edge
   "main_DB"."M"[26] := #_w19;
   IF #_w20 THEN "Z.H 7" := TRUE; END_IF;
   #_w21 := NOT #_w19 AND "main_DB"."M"[27];   // falling edge
   "main_DB"."M"[27] := #_w19;
   IF #_w21 THEN "Z.H 7" := FALSE; END_IF;
   #_w22 := "main_DB".Button.Screen_2."Z.H 8" AND "main_DB".Status.Manual_control;
   #_w23 := #_w22 AND NOT "main_DB"."M"[28];   // rising edge
   "main_DB"."M"[28] := #_w22;
   IF #_w23 THEN "Z.H 8" := TRUE; END_IF;
   #_w24 := NOT #_w22 AND "main_DB"."M"[29];   // falling edge
   "main_DB"."M"[29] := #_w22;
   IF #_w24 THEN "Z.H 8" := FALSE; END_IF;
END_REGION

REGION Network 12: "main_DB".var.Hydraulic_oil_pressure
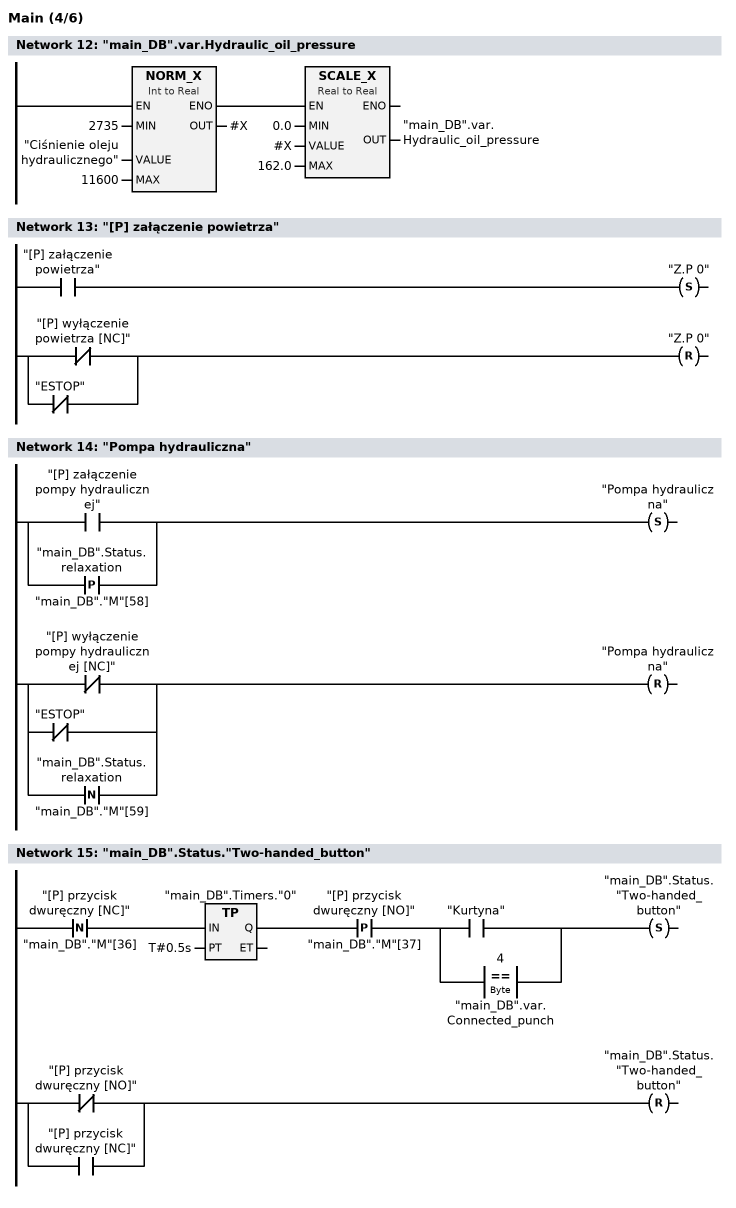
   RUNG wire#powerrail
      { S7_Templates := "[SrcType := Int, DestType := Real]" } Normalize(min := 2735, value := "Ciśnienie oleju hydraulicznego", max := 11600, out => #X)
      { S7_Templates := "[SrcType := Real, DestType := Real]" } Scale(min := 0.0, value := #X, max := 162.0, out => "main_DB".var.Hydraulic_oil_pressure)
   END_RUNG
   // the same network as SCL:
   #X := NORM_X(MIN := 2735, VALUE := "Ciśnienie oleju hydraulicznego", MAX := 11600);
   "main_DB".var.Hydraulic_oil_pressure := SCALE_X(MIN := 0.0, VALUE := #X, MAX := 162.0);
END_REGION

REGION Network 13: "[P] załączenie powietrza"
   RUNG wire#powerrail
      Contact( "[P] załączenie powietrza" )
      S_Coil( "Z.P 0" )
   END_RUNG
   RUNG wire#powerrail
      I_Contact( "[P] wyłączenie powietrza [NC]" )
      wire#w1
      R_Coil( "Z.P 0" )
   END_RUNG
   RUNG wire#powerrail
      I_Contact( "ESTOP" )
   END_RUNG wire#w1
   // the same network as SCL:
   IF "[P] załączenie powietrza" THEN "Z.P 0" := TRUE; END_IF;
   IF NOT "[P] wyłączenie powietrza [NC]" OR NOT "ESTOP" THEN "Z.P 0" := FALSE; END_IF;
END_REGION

REGION Network 14: "Pompa hydrauliczna"
   RUNG wire#powerrail
      Contact( "[P] załączenie pompy hydraulicznej" )
      wire#w1
      S_Coil( "Pompa hydrauliczna" )
   END_RUNG
   RUNG wire#powerrail
      P_Contact(operand := "main_DB".Status.relaxation, bit := "main_DB"."M"[58])
   END_RUNG wire#w1
   RUNG wire#powerrail
      I_Contact( "[P] wyłączenie pompy hydraulicznej [NC]" )
      wire#w2
      R_Coil( "Pompa hydrauliczna" )
   END_RUNG
   RUNG wire#powerrail
      I_Contact( "ESTOP" )
   END_RUNG wire#w2
   RUNG wire#powerrail
      N_Contact(operand := "main_DB".Status.relaxation, bit := "main_DB"."M"[59])
   END_RUNG wire#w2
   // the same network as SCL:
   #_w1 := "main_DB".Status.relaxation AND NOT "main_DB"."M"[58];   // rising edge of "main_DB".Status.relaxation
   "main_DB"."M"[58] := "main_DB".Status.relaxation;
   IF "[P] załączenie pompy hydraulicznej" OR #_w1 THEN "Pompa hydrauliczna" := TRUE; END_IF;
   #_w2 := NOT "main_DB".Status.relaxation AND "main_DB"."M"[59];   // falling edge of "main_DB".Status.relaxation
   "main_DB"."M"[59] := "main_DB".Status.relaxation;
   IF NOT "[P] wyłączenie pompy hydraulicznej [NC]" OR NOT "ESTOP" OR #_w2 THEN
       "Pompa hydrauliczna" := FALSE;
   END_IF;
END_REGION

REGION Network 15: "main_DB".Status."Two-handed_button"
   #_w1 := NOT "[P] przycisk dwuręczny [NC]" AND "main_DB"."M"[36];   // falling edge of "[P] przycisk dwuręczny [NC]"
   "main_DB"."M"[36] := "[P] przycisk dwuręczny [NC]";
   "main_DB".Timers."0".TP(IN := #_w1, PT := T#0.5s);
   #_w2 := "main_DB".Timers."0".Q AND "[P] przycisk dwuręczny [NO]" AND NOT "main_DB"."M"[37];   // rising edge of "[P] przycisk dwuręczny [NO]"
   "main_DB"."M"[37] := "[P] przycisk dwuręczny [NO]";
   IF #_w2 AND ("Kurtyna" OR (4 = "main_DB".var.Connected_punch)) THEN
       "main_DB".Status."Two-handed_button" := TRUE;
   END_IF;
   IF NOT "[P] przycisk dwuręczny [NO]" OR "[P] przycisk dwuręczny [NC]" THEN
       "main_DB".Status."Two-handed_button" := FALSE;
   END_IF;
END_REGION

REGION Network 16: Counters_reset
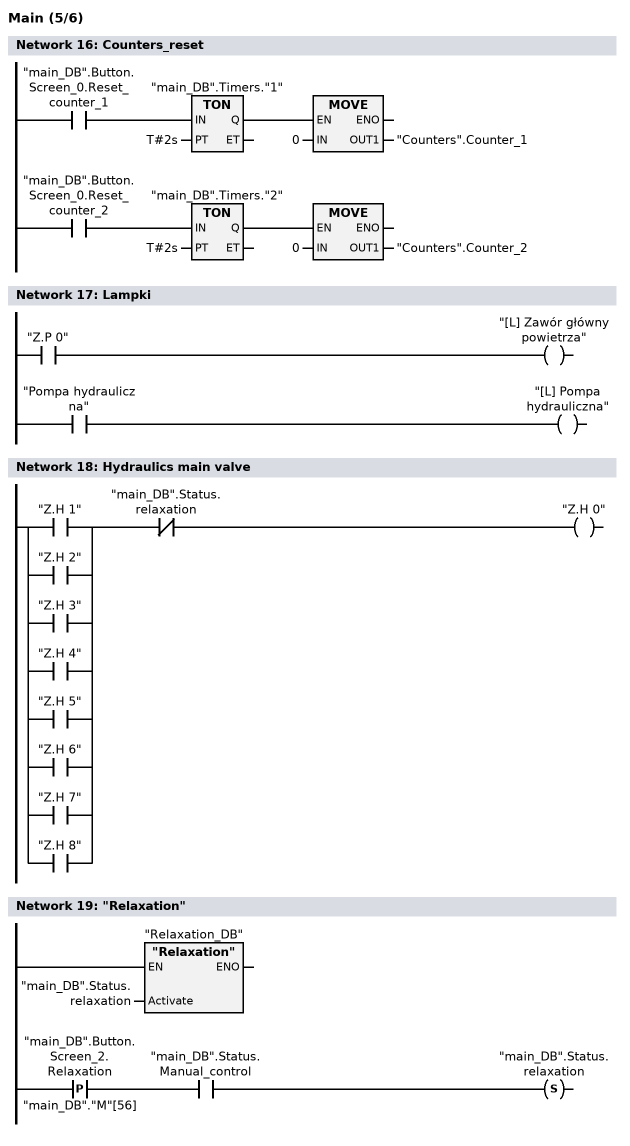
   "main_DB".Timers."1".TON(IN := "main_DB".Button.Screen_0.Reset_counter_1, PT := T#2s);
   IF "main_DB".Timers."1".Q THEN "Counters".Counter_1 := 0; END_IF;
   "main_DB".Timers."2".TON(IN := "main_DB".Button.Screen_0.Reset_counter_2, PT := T#2s);
   IF "main_DB".Timers."2".Q THEN "Counters".Counter_2 := 0; END_IF;
END_REGION

REGION Network 17: Lampki
   RUNG wire#powerrail
      Contact( "Z.P 0" )
      Coil( "[L] Zawór główny powietrza" )
   END_RUNG
   RUNG wire#powerrail
      Contact( "Pompa hydrauliczna" )
      Coil( "[L] Pompa hydrauliczna" )
   END_RUNG
   // the same network as SCL:
   "[L] Zawór główny powietrza" := "Z.P 0";
   "[L] Pompa hydrauliczna" := "Pompa hydrauliczna";
END_REGION

REGION Network 18: Hydraulics main valve
   RUNG wire#powerrail
      Contact( "Z.H 1" )
      wire#w1
      I_Contact( "main_DB".Status.relaxation )
      Coil( "Z.H 0" )
   END_RUNG
   RUNG wire#powerrail
      Contact( "Z.H 2" )
   END_RUNG wire#w1
   RUNG wire#powerrail
      Contact( "Z.H 3" )
   END_RUNG wire#w1
   RUNG wire#powerrail
      Contact( "Z.H 4" )
   END_RUNG wire#w1
   RUNG wire#powerrail
      Contact( "Z.H 5" )
   END_RUNG wire#w1
   RUNG wire#powerrail
      Contact( "Z.H 6" )
   END_RUNG wire#w1
   RUNG wire#powerrail
      Contact( "Z.H 7" )
   END_RUNG wire#w1
   RUNG wire#powerrail
      Contact( "Z.H 8" )
   END_RUNG wire#w1
   // the same network as SCL:
   "Z.H 0" := ("Z.H 1" OR "Z.H 2" OR "Z.H 3" OR "Z.H 4" OR "Z.H 5" OR "Z.H 6" OR "Z.H 7" OR "Z.H 8") AND NOT "main_DB".Status.relaxation;
END_REGION

REGION Network 19: "Relaxation"
   RUNG wire#powerrail
      "Relaxation_DB"(Activate := "main_DB".Status.relaxation)
   END_RUNG
   RUNG wire#powerrail
      P_Contact(operand := "main_DB".Button.Screen_2.Relaxation, bit := "main_DB"."M"[56])
      Contact( "main_DB".Status.Manual_control )
      S_Coil( "main_DB".Status.relaxation )
   END_RUNG
   // the same network as SCL:
   "Relaxation_DB"(Activate := "main_DB".Status.relaxation);   // "Relaxation"
   #_w1 := "main_DB".Button.Screen_2.Relaxation AND NOT "main_DB"."M"[56];   // rising edge of "main_DB".Button.Screen_2.Relaxation
   "main_DB"."M"[56] := "main_DB".Button.Screen_2.Relaxation;
   IF #_w1 AND "main_DB".Status.Manual_control THEN "main_DB".Status.relaxation := TRUE; END_IF;
END_REGION

REGION Network 20: Lubrication
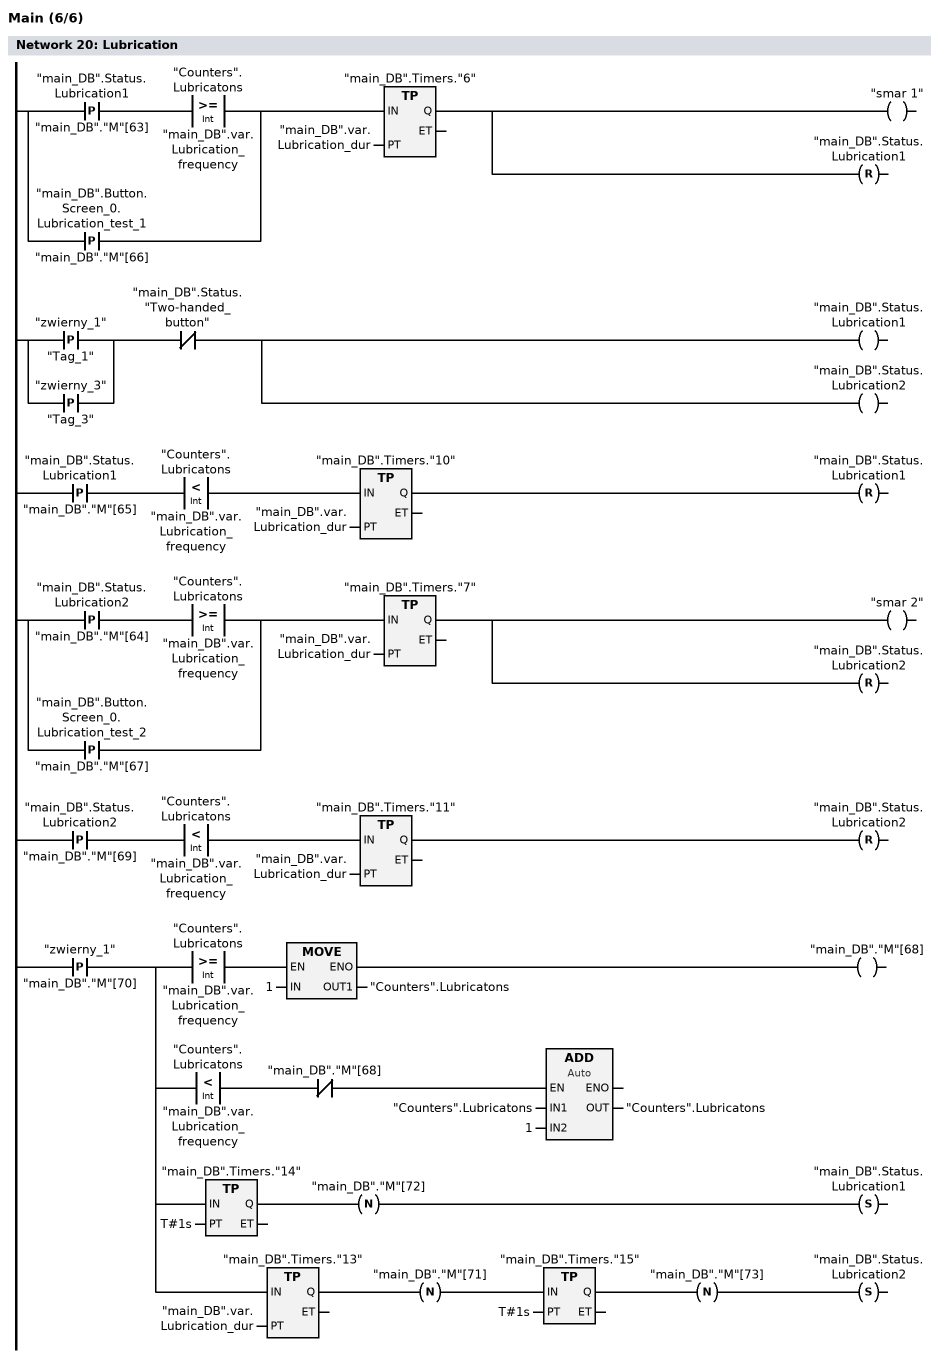
   #_w1 := "main_DB".Status.Lubrication1 AND NOT "main_DB"."M"[63];   // rising edge of "main_DB".Status.Lubrication1
   "main_DB"."M"[63] := "main_DB".Status.Lubrication1;
   #_w2 := "main_DB".Button.Screen_0.Lubrication_test_1 AND NOT "main_DB"."M"[66];   // rising edge of "main_DB".Button.Screen_0.Lubrication_test_1
   "main_DB"."M"[66] := "main_DB".Button.Screen_0.Lubrication_test_1;
   "main_DB".Timers."6".TP(IN := (#_w1 AND ("Counters".Lubricatons >= "main_DB".var.Lubrication_frequency)) OR #_w2,
                           PT := "main_DB".var.Lubrication_dur);
   "smar 1" := "main_DB".Timers."6".Q;
   IF "main_DB".Timers."6".Q THEN "main_DB".Status.Lubrication1 := FALSE; END_IF;
   #_w3 := "zwierny_1" AND NOT "Tag_1";   // rising edge of "zwierny_1"
   "Tag_1" := "zwierny_1";
   #_w4 := "zwierny_3" AND NOT "Tag_3";   // rising edge of "zwierny_3"
   "Tag_3" := "zwierny_3";
   "main_DB".Status.Lubrication1 := (#_w3 OR #_w4) AND NOT "main_DB".Status."Two-handed_button";
   "main_DB".Status.Lubrication2 := "main_DB".Status.Lubrication1;
   #_w5 := "main_DB".Status.Lubrication1 AND NOT "main_DB"."M"[65];   // rising edge of "main_DB".Status.Lubrication1
   "main_DB"."M"[65] := "main_DB".Status.Lubrication1;
   "main_DB".Timers."10".TP(IN := #_w5 AND ("Counters".Lubricatons < "main_DB".var.Lubrication_frequency),
                           PT := "main_DB".var.Lubrication_dur);
   IF "main_DB".Timers."10".Q THEN "main_DB".Status.Lubrication1 := FALSE; END_IF;
   #_w6 := "main_DB".Status.Lubrication2 AND NOT "main_DB"."M"[64];   // rising edge of "main_DB".Status.Lubrication2
   "main_DB"."M"[64] := "main_DB".Status.Lubrication2;
   #_w7 := "main_DB".Button.Screen_0.Lubrication_test_2 AND NOT "main_DB"."M"[67];   // rising edge of "main_DB".Button.Screen_0.Lubrication_test_2
   "main_DB"."M"[67] := "main_DB".Button.Screen_0.Lubrication_test_2;
   "main_DB".Timers."7".TP(IN := (#_w6 AND ("Counters".Lubricatons >= "main_DB".var.Lubrication_frequency)) OR #_w7,
                           PT := "main_DB".var.Lubrication_dur);
   "smar 2" := "main_DB".Timers."7".Q;
   IF "main_DB".Timers."7".Q THEN "main_DB".Status.Lubrication2 := FALSE; END_IF;
   #_w8 := "main_DB".Status.Lubrication2 AND NOT "main_DB"."M"[69];   // rising edge of "main_DB".Status.Lubrication2
   "main_DB"."M"[69] := "main_DB".Status.Lubrication2;
   "main_DB".Timers."11".TP(IN := #_w8 AND ("Counters".Lubricatons < "main_DB".var.Lubrication_frequency),
                           PT := "main_DB".var.Lubrication_dur);
   IF "main_DB".Timers."11".Q THEN "main_DB".Status.Lubrication2 := FALSE; END_IF;
   #_w9 := "zwierny_1" AND NOT "main_DB"."M"[70];   // rising edge of "zwierny_1"
   "main_DB"."M"[70] := "zwierny_1";
   #_w10 := #_w9 AND ("Counters".Lubricatons >= "main_DB".var.Lubrication_frequency);
   IF #_w10 THEN "Counters".Lubricatons := 1; END_IF;
   "main_DB"."M"[68] := #_w10;
   IF #_w9 AND ("Counters".Lubricatons < "main_DB".var.Lubrication_frequency) AND NOT "main_DB"."M"[68] THEN
       "Counters".Lubricatons := "Counters".Lubricatons + 1;
   END_IF;
   "main_DB".Timers."14".TP(IN := #_w9, PT := T#1s);
   #_w11 := NOT "main_DB".Timers."14".Q AND "main_DB"."M"[72];   // falling edge
   "main_DB"."M"[72] := "main_DB".Timers."14".Q;
   IF #_w11 THEN "main_DB".Status.Lubrication1 := TRUE; END_IF;
   "main_DB".Timers."13".TP(IN := #_w9, PT := "main_DB".var.Lubrication_dur);
   #_w12 := NOT "main_DB".Timers."13".Q AND "main_DB"."M"[71];   // falling edge
   "main_DB"."M"[71] := "main_DB".Timers."13".Q;
   "main_DB".Timers."15".TP(IN := #_w12, PT := T#1s);
   #_w13 := NOT "main_DB".Timers."15".Q AND "main_DB"."M"[73];   // falling edge
   "main_DB"."M"[73] := "main_DB".Timers."15".Q;
   IF #_w13 THEN "main_DB".Status.Lubrication2 := TRUE; END_IF;
END_REGION
END_ORGANIZATION_BLOCK

ORGANIZATION_BLOCK "Blink 100ms"   // OB30, LAD, CyclicInterrupt
{ S7_Optimized_Access := 'TRUE' }
VERSION : 0.1
   VAR_INPUT
      Initial_Call : Bool;   // Initial call of this OB
      Event_Count : Int;   // Events discarded
   END_VAR
BEGIN

REGION Network 1
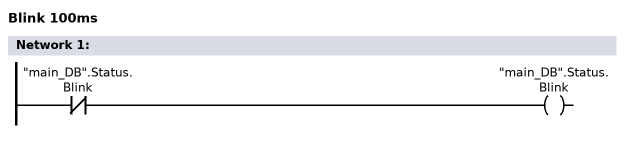
   RUNG wire#powerrail
      I_Contact( "main_DB".Status.Blink )
      Coil( "main_DB".Status.Blink )
   END_RUNG
   // the same network as SCL:
   "main_DB".Status.Blink := NOT "main_DB".Status.Blink;
END_REGION
END_ORGANIZATION_BLOCK

ORGANIZATION_BLOCK "Punch_parameters_rewrite"   // OB31, LAD, CyclicInterrupt
{ S7_Optimized_Access := 'TRUE' }
VERSION : 0.1
   VAR_INPUT
      Initial_Call : Bool;   // Initial call of this OB
      Event_Count : Int;   // Events discarded
   END_VAR
BEGIN

REGION Network 1 (SCL)
   "main_DB".var."Descryption Z.P 1" := "Punch_parameters".Punch["main_DB".var.Result_punch]."Z.P 1";
   "main_DB".var."Descryption Z.P 2" := "Punch_parameters".Punch["main_DB".var.Result_punch]."Z.P 2";
   "main_DB".var."Descryption Z.P 3" := "Punch_parameters".Punch["main_DB".var.Result_punch]."Z.P 3";
   "main_DB".var."Descryption Z.P 4" := "Punch_parameters".Punch["main_DB".var.Result_punch]."Z.P 4";

   "main_DB".var."Descryption Z.H 1" := "Punch_parameters".Punch["main_DB".var.Result_punch]."Z.H 1";
   "main_DB".var."Descryption Z.H 2" := "Punch_parameters".Punch["main_DB".var.Result_punch]."Z.H 2";
   "main_DB".var."Descryption Z.H 3" := "Punch_parameters".Punch["main_DB".var.Result_punch]."Z.H 3";
   "main_DB".var."Descryption Z.H 4" := "Punch_parameters".Punch["main_DB".var.Result_punch]."Z.H 4";
   "main_DB".var."Descryption Z.H 5" := "Punch_parameters".Punch["main_DB".var.Result_punch]."Z.H 5";
   "main_DB".var."Descryption Z.H 6" := "Punch_parameters".Punch["main_DB".var.Result_punch]."Z.H 6";
   "main_DB".var."Descryption Z.H 7" := "Punch_parameters".Punch["main_DB".var.Result_punch]."Z.H 7";
   "main_DB".var."Descryption Z.H 8" := "Punch_parameters".Punch["main_DB".var.Result_punch]."Z.H 8";

   "main_DB".var."Descryption SQ 1" := "Punch_parameters".Punch["main_DB".var.Result_punch].SQ1;
   "main_DB".var."Descryption SQ 2" := "Punch_parameters".Punch["main_DB".var.Result_punch].SQ2;
   "main_DB".var."Descryption SQ 3" := "Punch_parameters".Punch["main_DB".var.Result_punch].SQ3;
   "main_DB".var."Descryption SQ 4" := "Punch_parameters".Punch["main_DB".var.Result_punch].SQ4;
   "main_DB".var."Descryption SQ 5" := "Punch_parameters".Punch["main_DB".var.Result_punch].SQ5;
   "main_DB".var."Descryption SQ 6" := "Punch_parameters".Punch["main_DB".var.Result_punch].SQ6;

   "main_DB".var."Descryption contact_sensor 1" := "Punch_parameters".Punch["main_DB".var.Result_punch].Contact_sensor_1;
   "main_DB".var."Descryption contact_sensor 2" := "Punch_parameters".Punch["main_DB".var.Result_punch].Contact_sensor_2;
   "main_DB".var."Descryption contact_sensor 3" := "Punch_parameters".Punch["main_DB".var.Result_punch].Contact_sensor_3;
   "main_DB".var."Descryption contact_sensor 4" := "Punch_parameters".Punch["main_DB".var.Result_punch].Contact_sensor_4;
   "main_DB".var."Descryption contact_sensor 5" := "Punch_parameters".Punch["main_DB".var.Result_punch].Contact_sensor_5;
   "main_DB".var."Descryption contact_sensor 6" := "Punch_parameters".Punch["main_DB".var.Result_punch].Contact_sensor_6;
END_REGION

REGION Network 2 (SCL): Lubrication frequency
   IF "main_DB".var.Lubrication_frequency > 4 THEN
       "main_DB".var.Lubrication_frequency := 4;
       ;
   ELSIF "main_DB".var.Lubrication_frequency < 1 THEN
       "main_DB".var.Lubrication_frequency := 1;
       ;
   END_IF;
END_REGION
END_ORGANIZATION_BLOCK

// folder: Punch_blocks

FUNCTION_BLOCK "Punch1"   // FB1, LAD
{ S7_Optimized_Access := 'TRUE' }
VERSION : 0.1
   VAR_INPUT
      Active : Bool;
   END_VAR
   VAR
      finish : Bool;
      Cycle_time_overload : Bool;
   END_VAR
   VAR_TEMP
      In_cycle : Bool;
      ready : Bool;
   END_VAR
   VAR_TEMP   // added for the SCL form of the ladder/FBD networks
      _w1 : Bool;
      _w2 : Bool;
   END_VAR
BEGIN

REGION Network 1: #ready
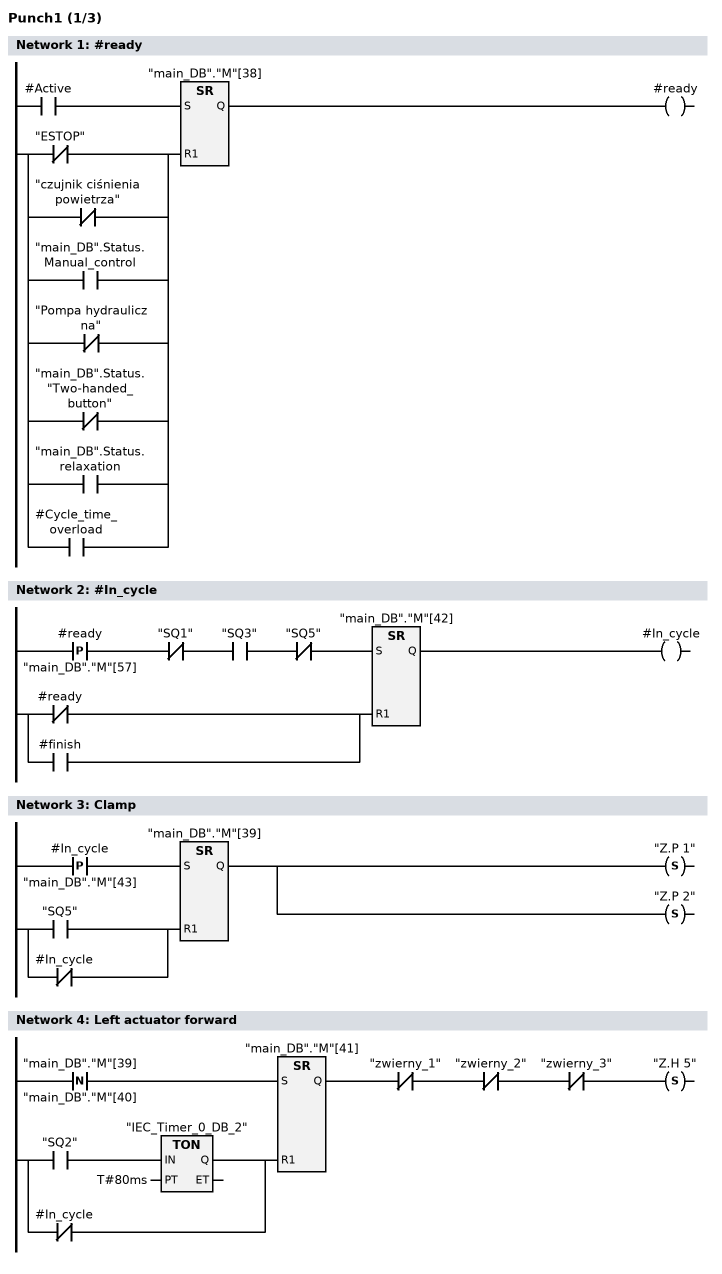
   RUNG wire#powerrail
      Contact( #Active )
      S_SR(operand := "main_DB"."M"[38], r1 := wire#w1)
      Coil( #ready )
   END_RUNG
   RUNG wire#powerrail
      I_Contact( "ESTOP" )
   END_RUNG wire#w1
   RUNG wire#powerrail
      I_Contact( "czujnik ciśnienia powietrza" )
   END_RUNG wire#w1
   RUNG wire#powerrail
      Contact( "main_DB".Status.Manual_control )
   END_RUNG wire#w1
   RUNG wire#powerrail
      I_Contact( "Pompa hydrauliczna" )
   END_RUNG wire#w1
   RUNG wire#powerrail
      I_Contact( "main_DB".Status."Two-handed_button" )
   END_RUNG wire#w1
   RUNG wire#powerrail
      Contact( "main_DB".Status.relaxation )
   END_RUNG wire#w1
   RUNG wire#powerrail
      Contact( #Cycle_time_overload )
   END_RUNG wire#w1
   // the same network as SCL:
   IF #Active THEN
       "main_DB"."M"[38] := TRUE;   // SR flip-flop
   END_IF;
   IF NOT "ESTOP" OR NOT "czujnik ciśnienia powietrza" OR "main_DB".Status.Manual_control OR NOT "Pompa hydrauliczna" OR NOT "main_DB".Status."Two-handed_button" OR "main_DB".Status.relaxation OR #Cycle_time_overload THEN
       "main_DB"."M"[38] := FALSE;
   END_IF;
   #ready := "main_DB"."M"[38];
END_REGION

REGION Network 2: #In_cycle
   RUNG wire#powerrail
      P_Contact(operand := #ready, bit := "main_DB"."M"[57])
      I_Contact( "SQ1" )
      Contact( "SQ3" )
      I_Contact( "SQ5" )
      S_SR(operand := "main_DB"."M"[42], r1 := wire#w1)
      Coil( #In_cycle )
   END_RUNG
   RUNG wire#powerrail
      I_Contact( #ready )
   END_RUNG wire#w1
   RUNG wire#powerrail
      Contact( #finish )
   END_RUNG wire#w1
   // the same network as SCL:
   #_w1 := #ready AND NOT "main_DB"."M"[57];   // rising edge of #ready
   "main_DB"."M"[57] := #ready;
   IF #_w1 AND NOT "SQ1" AND "SQ3" AND NOT "SQ5" THEN
       "main_DB"."M"[42] := TRUE;   // SR flip-flop
   END_IF;
   IF NOT #ready OR #finish THEN "main_DB"."M"[42] := FALSE; END_IF;
   #In_cycle := "main_DB"."M"[42];
END_REGION

REGION Network 3: Clamp
   RUNG wire#powerrail
      P_Contact(operand := #In_cycle, bit := "main_DB"."M"[43])
      S_SR(operand := "main_DB"."M"[39], r1 := wire#w1)
      wire#w2
      S_Coil( "Z.P 1" )
   END_RUNG
   RUNG wire#powerrail
      Contact( "SQ5" )
   END_RUNG wire#w1
   RUNG wire#powerrail
      I_Contact( #In_cycle )
   END_RUNG wire#w1
   RUNG wire#w2
      S_Coil( "Z.P 2" )
   END_RUNG
   // the same network as SCL:
   #_w1 := #In_cycle AND NOT "main_DB"."M"[43];   // rising edge of #In_cycle
   "main_DB"."M"[43] := #In_cycle;
   IF #_w1 THEN
       "main_DB"."M"[39] := TRUE;   // SR flip-flop
   END_IF;
   IF "SQ5" OR NOT #In_cycle THEN "main_DB"."M"[39] := FALSE; END_IF;
   IF "main_DB"."M"[39] THEN
       "Z.P 1" := TRUE;
       "Z.P 2" := TRUE;
   END_IF;
END_REGION

REGION Network 4: Left actuator forward
   #_w1 := NOT "main_DB"."M"[39] AND "main_DB"."M"[40];   // falling edge of "main_DB"."M"[39]
   "main_DB"."M"[40] := "main_DB"."M"[39];
   "IEC_Timer_0_DB_2".TON(IN := "SQ2", PT := T#80ms);
   IF #_w1 THEN
       "main_DB"."M"[41] := TRUE;   // SR flip-flop
   END_IF;
   IF "IEC_Timer_0_DB_2".Q OR NOT #In_cycle THEN "main_DB"."M"[41] := FALSE; END_IF;
   IF "main_DB"."M"[41] AND NOT "zwierny_1" AND NOT "zwierny_2" AND NOT "zwierny_3" THEN
       "Z.H 5" := TRUE;
   END_IF;
END_REGION

REGION Network 5: Right actuator forward
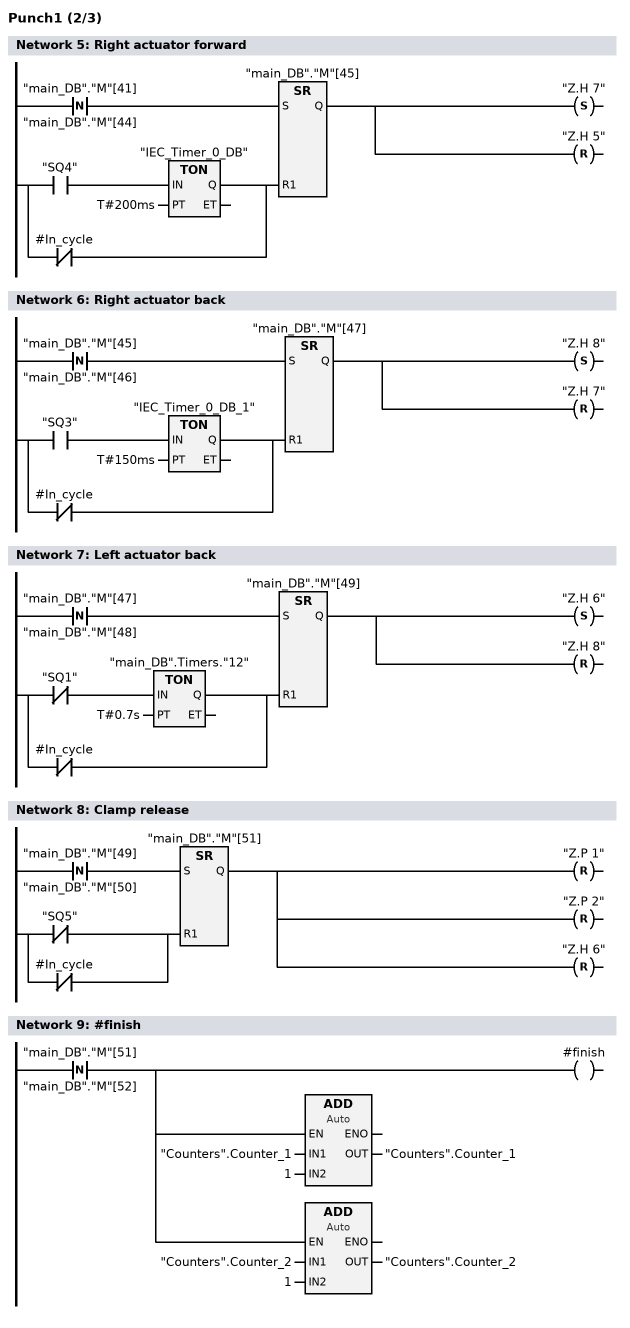
   #_w1 := NOT "main_DB"."M"[41] AND "main_DB"."M"[44];   // falling edge of "main_DB"."M"[41]
   "main_DB"."M"[44] := "main_DB"."M"[41];
   "IEC_Timer_0_DB".TON(IN := "SQ4", PT := T#200ms);
   IF #_w1 THEN
       "main_DB"."M"[45] := TRUE;   // SR flip-flop
   END_IF;
   IF "IEC_Timer_0_DB".Q OR NOT #In_cycle THEN "main_DB"."M"[45] := FALSE; END_IF;
   IF "main_DB"."M"[45] THEN
       "Z.H 7" := TRUE;
       "Z.H 5" := FALSE;
   END_IF;
END_REGION

REGION Network 6: Right actuator back
   #_w1 := NOT "main_DB"."M"[45] AND "main_DB"."M"[46];   // falling edge of "main_DB"."M"[45]
   "main_DB"."M"[46] := "main_DB"."M"[45];
   "IEC_Timer_0_DB_1".TON(IN := "SQ3", PT := T#150ms);
   IF #_w1 THEN
       "main_DB"."M"[47] := TRUE;   // SR flip-flop
   END_IF;
   IF "IEC_Timer_0_DB_1".Q OR NOT #In_cycle THEN "main_DB"."M"[47] := FALSE; END_IF;
   IF "main_DB"."M"[47] THEN
       "Z.H 8" := TRUE;
       "Z.H 7" := FALSE;
   END_IF;
END_REGION

REGION Network 7: Left actuator back
   #_w1 := NOT "main_DB"."M"[47] AND "main_DB"."M"[48];   // falling edge of "main_DB"."M"[47]
   "main_DB"."M"[48] := "main_DB"."M"[47];
   "main_DB".Timers."12".TON(IN := NOT "SQ1", PT := T#0.7s);
   IF #_w1 THEN
       "main_DB"."M"[49] := TRUE;   // SR flip-flop
   END_IF;
   IF "main_DB".Timers."12".Q OR NOT #In_cycle THEN "main_DB"."M"[49] := FALSE; END_IF;
   IF "main_DB"."M"[49] THEN
       "Z.H 6" := TRUE;
       "Z.H 8" := FALSE;
   END_IF;
END_REGION

REGION Network 8: Clamp release
   RUNG wire#powerrail
      N_Contact(operand := "main_DB"."M"[49], bit := "main_DB"."M"[50])
      S_SR(operand := "main_DB"."M"[51], r1 := wire#w1)
      wire#w2
      R_Coil( "Z.P 1" )
   END_RUNG
   RUNG wire#powerrail
      I_Contact( "SQ5" )
   END_RUNG wire#w1
   RUNG wire#powerrail
      I_Contact( #In_cycle )
   END_RUNG wire#w1
   RUNG wire#w2
      R_Coil( "Z.P 2" )
   END_RUNG
   RUNG wire#w2
      R_Coil( "Z.H 6" )
   END_RUNG
   // the same network as SCL:
   #_w1 := NOT "main_DB"."M"[49] AND "main_DB"."M"[50];   // falling edge of "main_DB"."M"[49]
   "main_DB"."M"[50] := "main_DB"."M"[49];
   IF #_w1 THEN
       "main_DB"."M"[51] := TRUE;   // SR flip-flop
   END_IF;
   IF NOT "SQ5" OR NOT #In_cycle THEN "main_DB"."M"[51] := FALSE; END_IF;
   IF "main_DB"."M"[51] THEN
       "Z.P 1" := FALSE;
       "Z.P 2" := FALSE;
       "Z.H 6" := FALSE;
   END_IF;
END_REGION

REGION Network 9: #finish
   RUNG wire#powerrail
      N_Contact(operand := "main_DB"."M"[51], bit := "main_DB"."M"[52])
      wire#w1
      Coil( #finish )
   END_RUNG
   RUNG wire#w1
      Add(in1 := "Counters".Counter_1, in2 := 1, out => "Counters".Counter_1)
   END_RUNG
   RUNG wire#w1
      Add(in1 := "Counters".Counter_2, in2 := 1, out => "Counters".Counter_2)
   END_RUNG
   // the same network as SCL:
   #_w1 := NOT "main_DB"."M"[51] AND "main_DB"."M"[52];   // falling edge of "main_DB"."M"[51]
   "main_DB"."M"[52] := "main_DB"."M"[51];
   #finish := #_w1;
   IF #_w1 THEN
       "Counters".Counter_1 := "Counters".Counter_1 + 1;
       "Counters".Counter_2 := "Counters".Counter_2 + 1;
   END_IF;
END_REGION

REGION Network 10: "Outputs_reset"
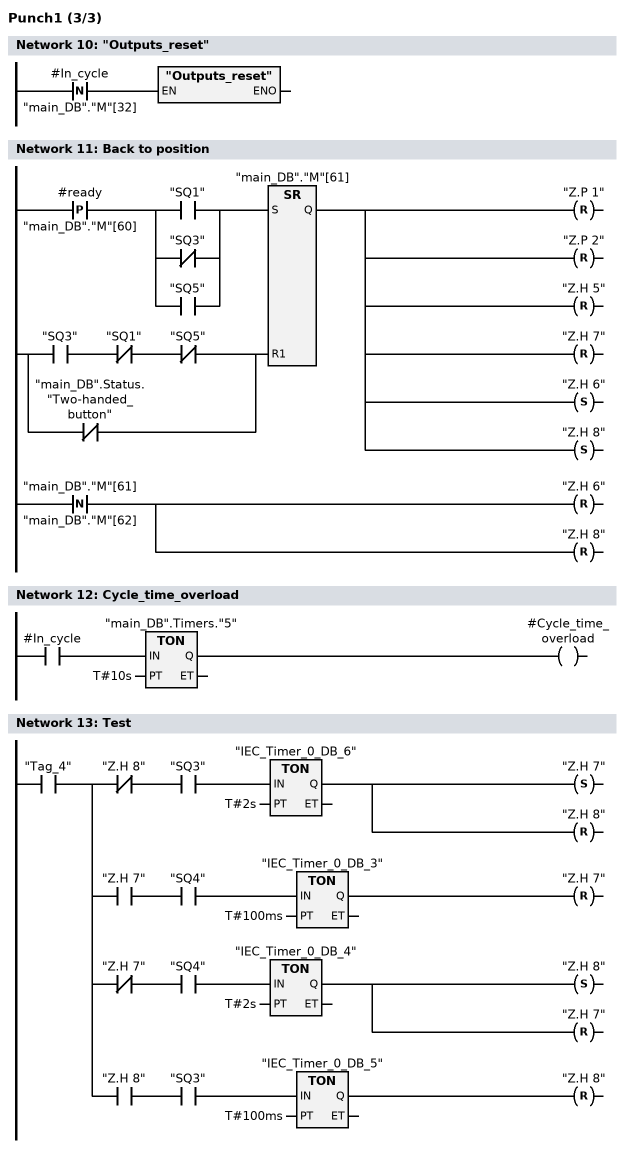
   RUNG wire#powerrail
      N_Contact(operand := #In_cycle, bit := "main_DB"."M"[32])
      "Outputs_reset"()
   END_RUNG
   // the same network as SCL:
   #_w1 := NOT #In_cycle AND "main_DB"."M"[32];   // falling edge of #In_cycle
   "main_DB"."M"[32] := #In_cycle;
   IF #_w1 THEN "Outputs_reset"(); END_IF;
END_REGION

REGION Network 11: Back to position
   RUNG wire#powerrail
      P_Contact(operand := #ready, bit := "main_DB"."M"[60])
      wire#w1
      Contact( "SQ1" )
      wire#w2
      S_SR(operand := "main_DB"."M"[61], r1 := wire#w3)
      wire#w4
      R_Coil( "Z.P 1" )
   END_RUNG
   RUNG wire#w1
      I_Contact( "SQ3" )
   END_RUNG wire#w2
   RUNG wire#w1
      Contact( "SQ5" )
   END_RUNG wire#w2
   RUNG wire#powerrail
      Contact( "SQ3" )
      I_Contact( "SQ1" )
      I_Contact( "SQ5" )
   END_RUNG wire#w3
   RUNG wire#powerrail
      I_Contact( "main_DB".Status."Two-handed_button" )
   END_RUNG wire#w3
   RUNG wire#w4
      R_Coil( "Z.P 2" )
   END_RUNG
   RUNG wire#w4
      R_Coil( "Z.H 5" )
   END_RUNG
   RUNG wire#w4
      R_Coil( "Z.H 7" )
   END_RUNG
   RUNG wire#w4
      S_Coil( "Z.H 6" )
   END_RUNG
   RUNG wire#w4
      S_Coil( "Z.H 8" )
   END_RUNG
   RUNG wire#powerrail
      N_Contact(operand := "main_DB"."M"[61], bit := "main_DB"."M"[62])
      wire#w5
      R_Coil( "Z.H 6" )
   END_RUNG
   RUNG wire#w5
      R_Coil( "Z.H 8" )
   END_RUNG
   // the same network as SCL:
   #_w1 := #ready AND NOT "main_DB"."M"[60];   // rising edge of #ready
   "main_DB"."M"[60] := #ready;
   IF #_w1 AND ("SQ1" OR NOT "SQ3" OR "SQ5") THEN
       "main_DB"."M"[61] := TRUE;   // SR flip-flop
   END_IF;
   IF ("SQ3" AND NOT "SQ1" AND NOT "SQ5") OR NOT "main_DB".Status."Two-handed_button" THEN
       "main_DB"."M"[61] := FALSE;
   END_IF;
   IF "main_DB"."M"[61] THEN
       "Z.P 1" := FALSE;
       "Z.P 2" := FALSE;
       "Z.H 5" := FALSE;
       "Z.H 7" := FALSE;
       "Z.H 6" := TRUE;
       "Z.H 8" := TRUE;
   END_IF;
   #_w2 := NOT "main_DB"."M"[61] AND "main_DB"."M"[62];   // falling edge of "main_DB"."M"[61]
   "main_DB"."M"[62] := "main_DB"."M"[61];
   IF #_w2 THEN
       "Z.H 6" := FALSE;
       "Z.H 8" := FALSE;
   END_IF;
END_REGION

REGION Network 12: Cycle_time_overload
   "main_DB".Timers."5".TON(IN := #In_cycle, PT := T#10s);
   #Cycle_time_overload := "main_DB".Timers."5".Q;
END_REGION

REGION Network 13: Test
   "IEC_Timer_0_DB_6".TON(IN := "Tag_4" AND NOT "Z.H 8" AND "SQ3", PT := T#2s);
   IF "IEC_Timer_0_DB_6".Q THEN
       "Z.H 7" := TRUE;
       "Z.H 8" := FALSE;
   END_IF;
   "IEC_Timer_0_DB_3".TON(IN := "Tag_4" AND "Z.H 7" AND "SQ4", PT := T#100ms);
   IF "IEC_Timer_0_DB_3".Q THEN "Z.H 7" := FALSE; END_IF;
   "IEC_Timer_0_DB_4".TON(IN := "Tag_4" AND NOT "Z.H 7" AND "SQ4", PT := T#2s);
   IF "IEC_Timer_0_DB_4".Q THEN
       "Z.H 8" := TRUE;
       "Z.H 7" := FALSE;
   END_IF;
   "IEC_Timer_0_DB_5".TON(IN := "Tag_4" AND "Z.H 8" AND "SQ3", PT := T#100ms);
   IF "IEC_Timer_0_DB_5".Q THEN "Z.H 8" := FALSE; END_IF;
END_REGION
END_FUNCTION_BLOCK

FUNCTION_BLOCK "Punch2"   // FB2, LAD
{ S7_Optimized_Access := 'TRUE' }
VERSION : 0.1
   VAR_INPUT
      Active : Bool;
   END_VAR
   VAR
      finish : Bool;
      Cycle_time_overload : Bool;
   END_VAR
   VAR_TEMP
      ready : Bool;
      In_cycle : Bool;
   END_VAR
   VAR_TEMP   // added for the SCL form of the ladder/FBD networks
      _w1 : Bool;
      _w2 : Bool;
   END_VAR
BEGIN

REGION Network 1: #ready
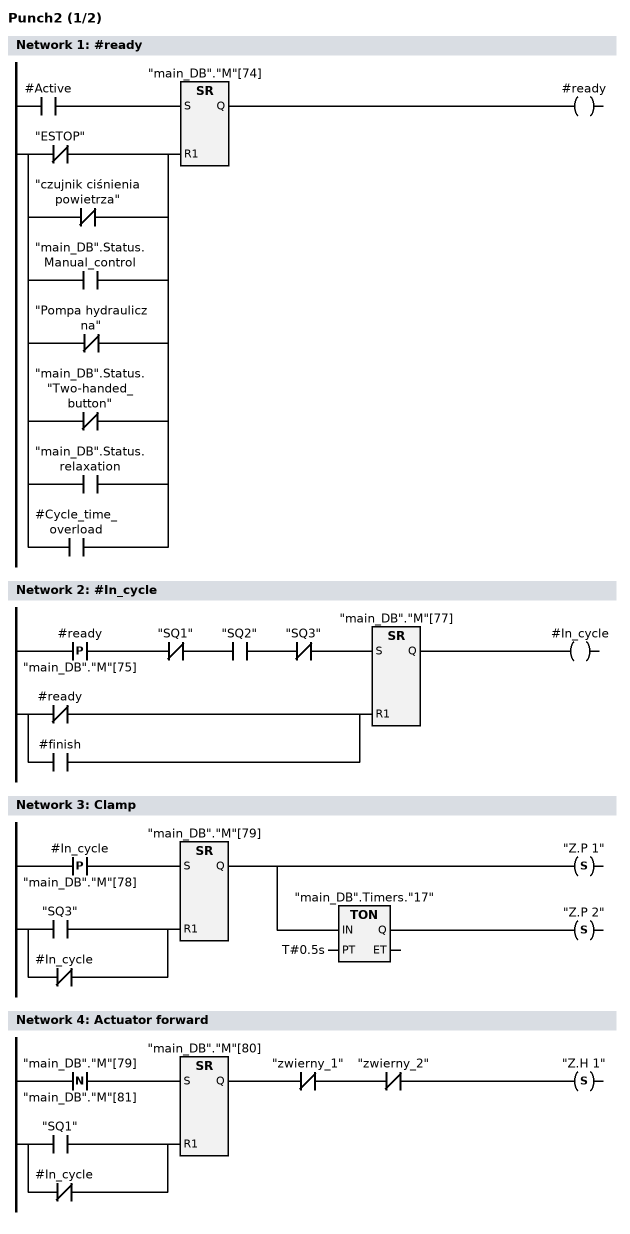
   RUNG wire#powerrail
      Contact( #Active )
      S_SR(operand := "main_DB"."M"[74], r1 := wire#w1)
      Coil( #ready )
   END_RUNG
   RUNG wire#powerrail
      I_Contact( "ESTOP" )
   END_RUNG wire#w1
   RUNG wire#powerrail
      I_Contact( "czujnik ciśnienia powietrza" )
   END_RUNG wire#w1
   RUNG wire#powerrail
      Contact( "main_DB".Status.Manual_control )
   END_RUNG wire#w1
   RUNG wire#powerrail
      I_Contact( "Pompa hydrauliczna" )
   END_RUNG wire#w1
   RUNG wire#powerrail
      I_Contact( "main_DB".Status."Two-handed_button" )
   END_RUNG wire#w1
   RUNG wire#powerrail
      Contact( "main_DB".Status.relaxation )
   END_RUNG wire#w1
   RUNG wire#powerrail
      Contact( #Cycle_time_overload )
   END_RUNG wire#w1
   // the same network as SCL:
   IF #Active THEN
       "main_DB"."M"[74] := TRUE;   // SR flip-flop
   END_IF;
   IF NOT "ESTOP" OR NOT "czujnik ciśnienia powietrza" OR "main_DB".Status.Manual_control OR NOT "Pompa hydrauliczna" OR NOT "main_DB".Status."Two-handed_button" OR "main_DB".Status.relaxation OR #Cycle_time_overload THEN
       "main_DB"."M"[74] := FALSE;
   END_IF;
   #ready := "main_DB"."M"[74];
END_REGION

REGION Network 2: #In_cycle
   RUNG wire#powerrail
      P_Contact(operand := #ready, bit := "main_DB"."M"[75])
      I_Contact( "SQ1" )
      Contact( "SQ2" )
      I_Contact( "SQ3" )
      S_SR(operand := "main_DB"."M"[77], r1 := wire#w1)
      Coil( #In_cycle )
   END_RUNG
   RUNG wire#powerrail
      I_Contact( #ready )
   END_RUNG wire#w1
   RUNG wire#powerrail
      Contact( #finish )
   END_RUNG wire#w1
   // the same network as SCL:
   #_w1 := #ready AND NOT "main_DB"."M"[75];   // rising edge of #ready
   "main_DB"."M"[75] := #ready;
   IF #_w1 AND NOT "SQ1" AND "SQ2" AND NOT "SQ3" THEN
       "main_DB"."M"[77] := TRUE;   // SR flip-flop
   END_IF;
   IF NOT #ready OR #finish THEN "main_DB"."M"[77] := FALSE; END_IF;
   #In_cycle := "main_DB"."M"[77];
END_REGION

REGION Network 3: Clamp
   #_w1 := #In_cycle AND NOT "main_DB"."M"[78];   // rising edge of #In_cycle
   "main_DB"."M"[78] := #In_cycle;
   IF #_w1 THEN
       "main_DB"."M"[79] := TRUE;   // SR flip-flop
   END_IF;
   IF "SQ3" OR NOT #In_cycle THEN "main_DB"."M"[79] := FALSE; END_IF;
   IF "main_DB"."M"[79] THEN "Z.P 1" := TRUE; END_IF;
   "main_DB".Timers."17".TON(IN := "main_DB"."M"[79], PT := T#0.5s);
   IF "main_DB".Timers."17".Q THEN "Z.P 2" := TRUE; END_IF;
END_REGION

REGION Network 4: Actuator forward
   RUNG wire#powerrail
      N_Contact(operand := "main_DB"."M"[79], bit := "main_DB"."M"[81])
      S_SR(operand := "main_DB"."M"[80], r1 := wire#w1)
      I_Contact( "zwierny_1" )
      I_Contact( "zwierny_2" )
      S_Coil( "Z.H 1" )
   END_RUNG
   RUNG wire#powerrail
      Contact( "SQ1" )
   END_RUNG wire#w1
   RUNG wire#powerrail
      I_Contact( #In_cycle )
   END_RUNG wire#w1
   // the same network as SCL:
   #_w1 := NOT "main_DB"."M"[79] AND "main_DB"."M"[81];   // falling edge of "main_DB"."M"[79]
   "main_DB"."M"[81] := "main_DB"."M"[79];
   IF #_w1 THEN
       "main_DB"."M"[80] := TRUE;   // SR flip-flop
   END_IF;
   IF "SQ1" OR NOT #In_cycle THEN "main_DB"."M"[80] := FALSE; END_IF;
   IF "main_DB"."M"[80] AND NOT "zwierny_1" AND NOT "zwierny_2" THEN "Z.H 1" := TRUE; END_IF;
END_REGION

REGION Network 5: Actuator back
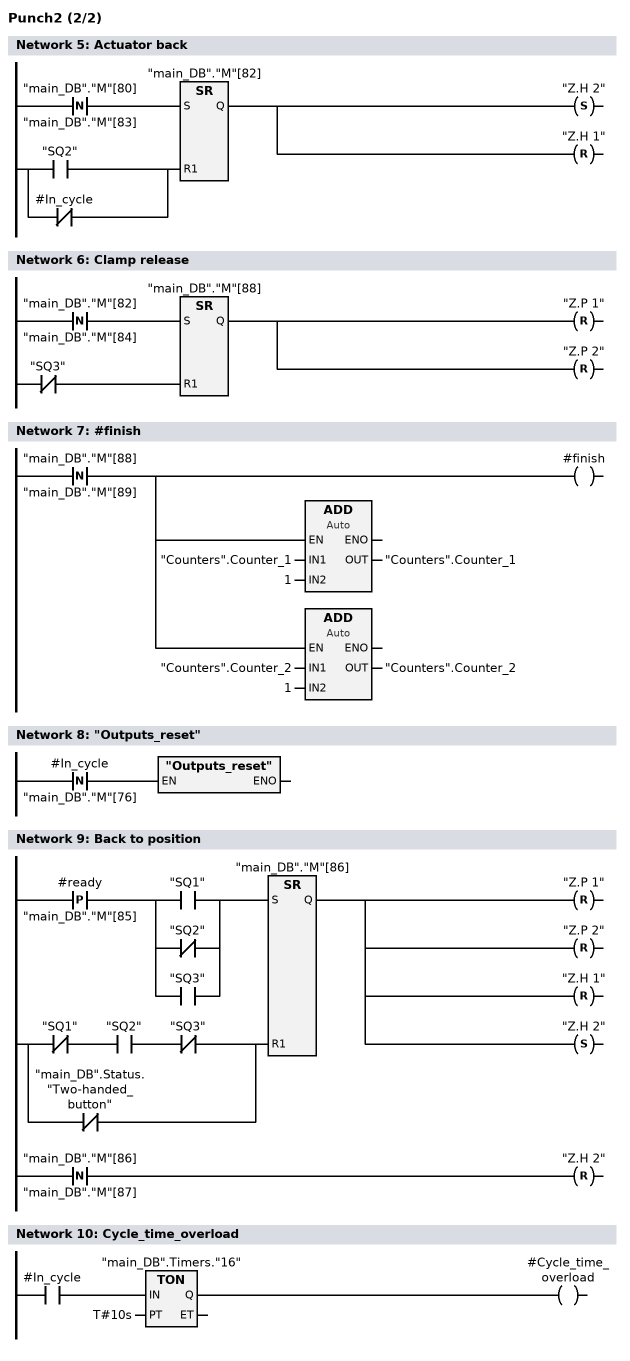
   RUNG wire#powerrail
      N_Contact(operand := "main_DB"."M"[80], bit := "main_DB"."M"[83])
      S_SR(operand := "main_DB"."M"[82], r1 := wire#w1)
      wire#w2
      S_Coil( "Z.H 2" )
   END_RUNG
   RUNG wire#powerrail
      Contact( "SQ2" )
   END_RUNG wire#w1
   RUNG wire#powerrail
      I_Contact( #In_cycle )
   END_RUNG wire#w1
   RUNG wire#w2
      R_Coil( "Z.H 1" )
   END_RUNG
   // the same network as SCL:
   #_w1 := NOT "main_DB"."M"[80] AND "main_DB"."M"[83];   // falling edge of "main_DB"."M"[80]
   "main_DB"."M"[83] := "main_DB"."M"[80];
   IF #_w1 THEN
       "main_DB"."M"[82] := TRUE;   // SR flip-flop
   END_IF;
   IF "SQ2" OR NOT #In_cycle THEN "main_DB"."M"[82] := FALSE; END_IF;
   IF "main_DB"."M"[82] THEN
       "Z.H 2" := TRUE;
       "Z.H 1" := FALSE;
   END_IF;
END_REGION

REGION Network 6: Clamp release
   RUNG wire#powerrail
      N_Contact(operand := "main_DB"."M"[82], bit := "main_DB"."M"[84])
      S_SR(operand := "main_DB"."M"[88], r1 := wire#w1)
      wire#w2
      R_Coil( "Z.P 1" )
   END_RUNG
   RUNG wire#powerrail
      I_Contact( "SQ3" )
   END_RUNG wire#w1
   RUNG wire#w2
      R_Coil( "Z.P 2" )
   END_RUNG
   // the same network as SCL:
   #_w1 := NOT "main_DB"."M"[82] AND "main_DB"."M"[84];   // falling edge of "main_DB"."M"[82]
   "main_DB"."M"[84] := "main_DB"."M"[82];
   IF #_w1 THEN
       "main_DB"."M"[88] := TRUE;   // SR flip-flop
   END_IF;
   IF NOT "SQ3" THEN "main_DB"."M"[88] := FALSE; END_IF;
   IF "main_DB"."M"[88] THEN
       "Z.P 1" := FALSE;
       "Z.P 2" := FALSE;
   END_IF;
END_REGION

REGION Network 7: #finish
   RUNG wire#powerrail
      N_Contact(operand := "main_DB"."M"[88], bit := "main_DB"."M"[89])
      wire#w1
      Coil( #finish )
   END_RUNG
   RUNG wire#w1
      Add(in1 := "Counters".Counter_1, in2 := 1, out => "Counters".Counter_1)
   END_RUNG
   RUNG wire#w1
      Add(in1 := "Counters".Counter_2, in2 := 1, out => "Counters".Counter_2)
   END_RUNG
   // the same network as SCL:
   #_w1 := NOT "main_DB"."M"[88] AND "main_DB"."M"[89];   // falling edge of "main_DB"."M"[88]
   "main_DB"."M"[89] := "main_DB"."M"[88];
   #finish := #_w1;
   IF #_w1 THEN
       "Counters".Counter_1 := "Counters".Counter_1 + 1;
       "Counters".Counter_2 := "Counters".Counter_2 + 1;
   END_IF;
END_REGION

REGION Network 8: "Outputs_reset"
   RUNG wire#powerrail
      N_Contact(operand := #In_cycle, bit := "main_DB"."M"[76])
      "Outputs_reset"()
   END_RUNG
   // the same network as SCL:
   #_w1 := NOT #In_cycle AND "main_DB"."M"[76];   // falling edge of #In_cycle
   "main_DB"."M"[76] := #In_cycle;
   IF #_w1 THEN "Outputs_reset"(); END_IF;
END_REGION

REGION Network 9: Back to position
   RUNG wire#powerrail
      P_Contact(operand := #ready, bit := "main_DB"."M"[85])
      wire#w1
      Contact( "SQ1" )
      wire#w2
      S_SR(operand := "main_DB"."M"[86], r1 := wire#w3)
      wire#w4
      R_Coil( "Z.P 1" )
   END_RUNG
   RUNG wire#w1
      I_Contact( "SQ2" )
   END_RUNG wire#w2
   RUNG wire#w1
      Contact( "SQ3" )
   END_RUNG wire#w2
   RUNG wire#powerrail
      I_Contact( "SQ1" )
      Contact( "SQ2" )
      I_Contact( "SQ3" )
   END_RUNG wire#w3
   RUNG wire#powerrail
      I_Contact( "main_DB".Status."Two-handed_button" )
   END_RUNG wire#w3
   RUNG wire#w4
      R_Coil( "Z.P 2" )
   END_RUNG
   RUNG wire#w4
      R_Coil( "Z.H 1" )
   END_RUNG
   RUNG wire#w4
      S_Coil( "Z.H 2" )
   END_RUNG
   RUNG wire#powerrail
      N_Contact(operand := "main_DB"."M"[86], bit := "main_DB"."M"[87])
      R_Coil( "Z.H 2" )
   END_RUNG
   // the same network as SCL:
   #_w1 := #ready AND NOT "main_DB"."M"[85];   // rising edge of #ready
   "main_DB"."M"[85] := #ready;
   IF #_w1 AND ("SQ1" OR NOT "SQ2" OR "SQ3") THEN
       "main_DB"."M"[86] := TRUE;   // SR flip-flop
   END_IF;
   IF (NOT "SQ1" AND "SQ2" AND NOT "SQ3") OR NOT "main_DB".Status."Two-handed_button" THEN
       "main_DB"."M"[86] := FALSE;
   END_IF;
   IF "main_DB"."M"[86] THEN
       "Z.P 1" := FALSE;
       "Z.P 2" := FALSE;
       "Z.H 1" := FALSE;
       "Z.H 2" := TRUE;
   END_IF;
   #_w2 := NOT "main_DB"."M"[86] AND "main_DB"."M"[87];   // falling edge of "main_DB"."M"[86]
   "main_DB"."M"[87] := "main_DB"."M"[86];
   IF #_w2 THEN "Z.H 2" := FALSE; END_IF;
END_REGION

REGION Network 10: Cycle_time_overload
   "main_DB".Timers."16".TON(IN := #In_cycle, PT := T#10s);
   #Cycle_time_overload := "main_DB".Timers."16".Q;
END_REGION
END_FUNCTION_BLOCK

FUNCTION_BLOCK "Punch3"   // FB3, LAD
{ S7_Optimized_Access := 'TRUE' }
VERSION : 0.1
   VAR_INPUT
      Active : Bool;
   END_VAR
   VAR
      finish : Bool;
      Back_to_pos : Bool;
      finishing : Bool;
      Cycle_time_overload : Bool;
   END_VAR
   VAR_TEMP
      In_cycle : Bool;
      ready : Bool;
   END_VAR
   VAR_TEMP   // added for the SCL form of the ladder/FBD networks
      _w1 : Bool;
      _w2 : Bool;
   END_VAR
BEGIN

REGION Network 1: #ready
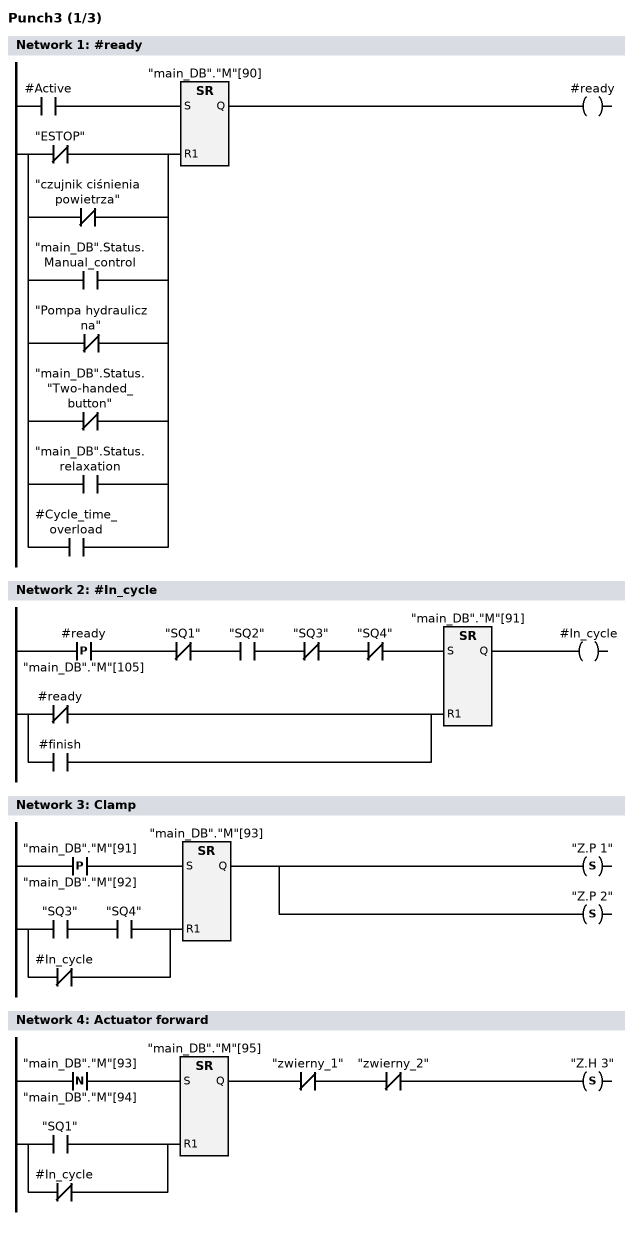
   RUNG wire#powerrail
      Contact( #Active )
      S_SR(operand := "main_DB"."M"[90], r1 := wire#w1)
      Coil( #ready )
   END_RUNG
   RUNG wire#powerrail
      I_Contact( "ESTOP" )
   END_RUNG wire#w1
   RUNG wire#powerrail
      I_Contact( "czujnik ciśnienia powietrza" )
   END_RUNG wire#w1
   RUNG wire#powerrail
      Contact( "main_DB".Status.Manual_control )
   END_RUNG wire#w1
   RUNG wire#powerrail
      I_Contact( "Pompa hydrauliczna" )
   END_RUNG wire#w1
   RUNG wire#powerrail
      I_Contact( "main_DB".Status."Two-handed_button" )
   END_RUNG wire#w1
   RUNG wire#powerrail
      Contact( "main_DB".Status.relaxation )
   END_RUNG wire#w1
   RUNG wire#powerrail
      Contact( #Cycle_time_overload )
   END_RUNG wire#w1
   // the same network as SCL:
   IF #Active THEN
       "main_DB"."M"[90] := TRUE;   // SR flip-flop
   END_IF;
   IF NOT "ESTOP" OR NOT "czujnik ciśnienia powietrza" OR "main_DB".Status.Manual_control OR NOT "Pompa hydrauliczna" OR NOT "main_DB".Status."Two-handed_button" OR "main_DB".Status.relaxation OR #Cycle_time_overload THEN
       "main_DB"."M"[90] := FALSE;
   END_IF;
   #ready := "main_DB"."M"[90];
END_REGION

REGION Network 2: #In_cycle
   RUNG wire#powerrail
      P_Contact(operand := #ready, bit := "main_DB"."M"[105])
      I_Contact( "SQ1" )
      Contact( "SQ2" )
      I_Contact( "SQ3" )
      I_Contact( "SQ4" )
      S_SR(operand := "main_DB"."M"[91], r1 := wire#w1)
      Coil( #In_cycle )
   END_RUNG
   RUNG wire#powerrail
      I_Contact( #ready )
   END_RUNG wire#w1
   RUNG wire#powerrail
      Contact( #finish )
   END_RUNG wire#w1
   // the same network as SCL:
   #_w1 := #ready AND NOT "main_DB"."M"[105];   // rising edge of #ready
   "main_DB"."M"[105] := #ready;
   IF #_w1 AND NOT "SQ1" AND "SQ2" AND NOT "SQ3" AND NOT "SQ4" THEN
       "main_DB"."M"[91] := TRUE;   // SR flip-flop
   END_IF;
   IF NOT #ready OR #finish THEN "main_DB"."M"[91] := FALSE; END_IF;
   #In_cycle := "main_DB"."M"[91];
END_REGION

REGION Network 3: Clamp
   RUNG wire#powerrail
      P_Contact(operand := "main_DB"."M"[91], bit := "main_DB"."M"[92])
      S_SR(operand := "main_DB"."M"[93], r1 := wire#w1)
      wire#w2
      S_Coil( "Z.P 1" )
   END_RUNG
   RUNG wire#powerrail
      Contact( "SQ3" )
      Contact( "SQ4" )
   END_RUNG wire#w1
   RUNG wire#powerrail
      I_Contact( #In_cycle )
   END_RUNG wire#w1
   RUNG wire#w2
      S_Coil( "Z.P 2" )
   END_RUNG
   // the same network as SCL:
   #_w1 := "main_DB"."M"[91] AND NOT "main_DB"."M"[92];   // rising edge of "main_DB"."M"[91]
   "main_DB"."M"[92] := "main_DB"."M"[91];
   IF #_w1 THEN
       "main_DB"."M"[93] := TRUE;   // SR flip-flop
   END_IF;
   IF ("SQ3" AND "SQ4") OR NOT #In_cycle THEN "main_DB"."M"[93] := FALSE; END_IF;
   IF "main_DB"."M"[93] THEN
       "Z.P 1" := TRUE;
       "Z.P 2" := TRUE;
   END_IF;
END_REGION

REGION Network 4: Actuator forward
   RUNG wire#powerrail
      N_Contact(operand := "main_DB"."M"[93], bit := "main_DB"."M"[94])
      S_SR(operand := "main_DB"."M"[95], r1 := wire#w1)
      I_Contact( "zwierny_1" )
      I_Contact( "zwierny_2" )
      S_Coil( "Z.H 3" )
   END_RUNG
   RUNG wire#powerrail
      Contact( "SQ1" )
   END_RUNG wire#w1
   RUNG wire#powerrail
      I_Contact( #In_cycle )
   END_RUNG wire#w1
   // the same network as SCL:
   #_w1 := NOT "main_DB"."M"[93] AND "main_DB"."M"[94];   // falling edge of "main_DB"."M"[93]
   "main_DB"."M"[94] := "main_DB"."M"[93];
   IF #_w1 THEN
       "main_DB"."M"[95] := TRUE;   // SR flip-flop
   END_IF;
   IF "SQ1" OR NOT #In_cycle THEN "main_DB"."M"[95] := FALSE; END_IF;
   IF "main_DB"."M"[95] AND NOT "zwierny_1" AND NOT "zwierny_2" THEN "Z.H 3" := TRUE; END_IF;
END_REGION

REGION Network 5: Actuator back
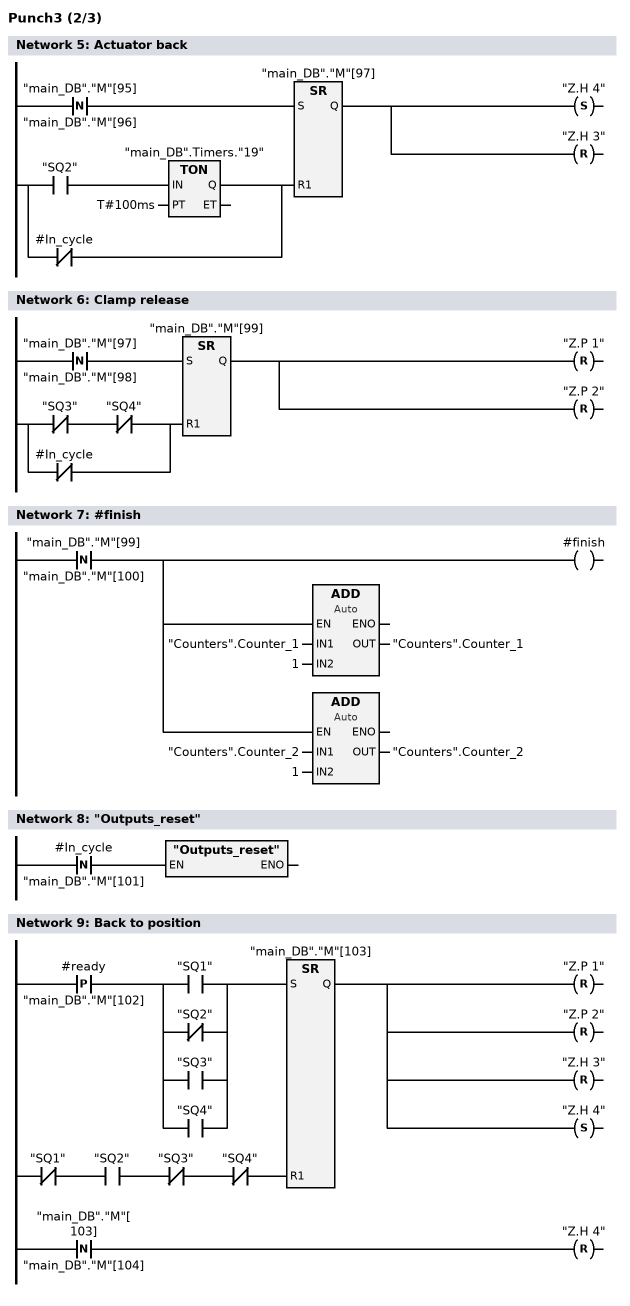
   #_w1 := NOT "main_DB"."M"[95] AND "main_DB"."M"[96];   // falling edge of "main_DB"."M"[95]
   "main_DB"."M"[96] := "main_DB"."M"[95];
   "main_DB".Timers."19".TON(IN := "SQ2", PT := T#100ms);
   IF #_w1 THEN
       "main_DB"."M"[97] := TRUE;   // SR flip-flop
   END_IF;
   IF "main_DB".Timers."19".Q OR NOT #In_cycle THEN "main_DB"."M"[97] := FALSE; END_IF;
   IF "main_DB"."M"[97] THEN
       "Z.H 4" := TRUE;
       "Z.H 3" := FALSE;
   END_IF;
END_REGION

REGION Network 6: Clamp release
   RUNG wire#powerrail
      N_Contact(operand := "main_DB"."M"[97], bit := "main_DB"."M"[98])
      S_SR(operand := "main_DB"."M"[99], r1 := wire#w1)
      wire#w2
      R_Coil( "Z.P 1" )
   END_RUNG
   RUNG wire#powerrail
      I_Contact( "SQ3" )
      I_Contact( "SQ4" )
   END_RUNG wire#w1
   RUNG wire#powerrail
      I_Contact( #In_cycle )
   END_RUNG wire#w1
   RUNG wire#w2
      R_Coil( "Z.P 2" )
   END_RUNG
   // the same network as SCL:
   #_w1 := NOT "main_DB"."M"[97] AND "main_DB"."M"[98];   // falling edge of "main_DB"."M"[97]
   "main_DB"."M"[98] := "main_DB"."M"[97];
   IF #_w1 THEN
       "main_DB"."M"[99] := TRUE;   // SR flip-flop
   END_IF;
   IF (NOT "SQ3" AND NOT "SQ4") OR NOT #In_cycle THEN "main_DB"."M"[99] := FALSE; END_IF;
   IF "main_DB"."M"[99] THEN
       "Z.P 1" := FALSE;
       "Z.P 2" := FALSE;
   END_IF;
END_REGION

REGION Network 7: #finish
   RUNG wire#powerrail
      N_Contact(operand := "main_DB"."M"[99], bit := "main_DB"."M"[100])
      wire#w1
      Coil( #finish )
   END_RUNG
   RUNG wire#w1
      Add(in1 := "Counters".Counter_1, in2 := 1, out => "Counters".Counter_1)
   END_RUNG
   RUNG wire#w1
      Add(in1 := "Counters".Counter_2, in2 := 1, out => "Counters".Counter_2)
   END_RUNG
   // the same network as SCL:
   #_w1 := NOT "main_DB"."M"[99] AND "main_DB"."M"[100];   // falling edge of "main_DB"."M"[99]
   "main_DB"."M"[100] := "main_DB"."M"[99];
   #finish := #_w1;
   IF #_w1 THEN
       "Counters".Counter_1 := "Counters".Counter_1 + 1;
       "Counters".Counter_2 := "Counters".Counter_2 + 1;
   END_IF;
END_REGION

REGION Network 8: "Outputs_reset"
   RUNG wire#powerrail
      N_Contact(operand := #In_cycle, bit := "main_DB"."M"[101])
      "Outputs_reset"()
   END_RUNG
   // the same network as SCL:
   #_w1 := NOT #In_cycle AND "main_DB"."M"[101];   // falling edge of #In_cycle
   "main_DB"."M"[101] := #In_cycle;
   IF #_w1 THEN "Outputs_reset"(); END_IF;
END_REGION

REGION Network 9: Back to position
   RUNG wire#powerrail
      P_Contact(operand := #ready, bit := "main_DB"."M"[102])
      wire#w1
      Contact( "SQ1" )
      wire#w2
      S_SR(operand := "main_DB"."M"[103], r1 := wire#w3)
      wire#w4
      R_Coil( "Z.P 1" )
   END_RUNG
   RUNG wire#w1
      I_Contact( "SQ2" )
   END_RUNG wire#w2
   RUNG wire#w1
      Contact( "SQ3" )
   END_RUNG wire#w2
   RUNG wire#w1
      Contact( "SQ4" )
   END_RUNG wire#w2
   RUNG wire#powerrail
      I_Contact( "SQ1" )
      Contact( "SQ2" )
      I_Contact( "SQ3" )
      I_Contact( "SQ4" )
   END_RUNG wire#w3
   RUNG wire#w4
      R_Coil( "Z.P 2" )
   END_RUNG
   RUNG wire#w4
      R_Coil( "Z.H 3" )
   END_RUNG
   RUNG wire#w4
      S_Coil( "Z.H 4" )
   END_RUNG
   RUNG wire#powerrail
      N_Contact(operand := "main_DB"."M"[103], bit := "main_DB"."M"[104])
      R_Coil( "Z.H 4" )
   END_RUNG
   // the same network as SCL:
   #_w1 := #ready AND NOT "main_DB"."M"[102];   // rising edge of #ready
   "main_DB"."M"[102] := #ready;
   IF #_w1 AND ("SQ1" OR NOT "SQ2" OR "SQ3" OR "SQ4") THEN
       "main_DB"."M"[103] := TRUE;   // SR flip-flop
   END_IF;
   IF NOT "SQ1" AND "SQ2" AND NOT "SQ3" AND NOT "SQ4" THEN "main_DB"."M"[103] := FALSE; END_IF;
   IF "main_DB"."M"[103] THEN
       "Z.P 1" := FALSE;
       "Z.P 2" := FALSE;
       "Z.H 3" := FALSE;
       "Z.H 4" := TRUE;
   END_IF;
   #_w2 := NOT "main_DB"."M"[103] AND "main_DB"."M"[104];   // falling edge of "main_DB"."M"[103]
   "main_DB"."M"[104] := "main_DB"."M"[103];
   IF #_w2 THEN "Z.H 4" := FALSE; END_IF;
END_REGION

REGION Network 10: Cycle_time_overload
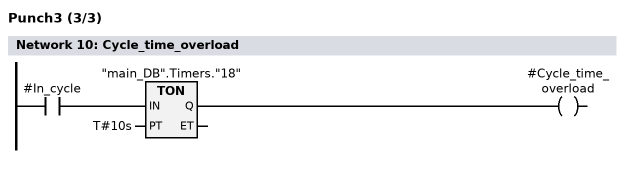
   "main_DB".Timers."18".TON(IN := #In_cycle, PT := T#10s);
   #Cycle_time_overload := "main_DB".Timers."18".Q;
END_REGION
END_FUNCTION_BLOCK

FUNCTION_BLOCK "Punch4"   // FB5, LAD
{ S7_Optimized_Access := 'TRUE' }
VERSION : 0.1
   VAR_INPUT
      Active : Bool;
   END_VAR
   VAR
      finish : Bool;
      Punching_finished_sum : Bool;
      Cycle_time_overload : Bool;
   END_VAR
   VAR_TEMP
      In_cycle : Bool;
      ready : Bool;
   END_VAR
   VAR_TEMP   // added for the SCL form of the ladder/FBD networks
      _w1 : Bool;
      _w2 : Bool;
      _w3 : Bool;
   END_VAR
BEGIN

REGION Network 1: #ready
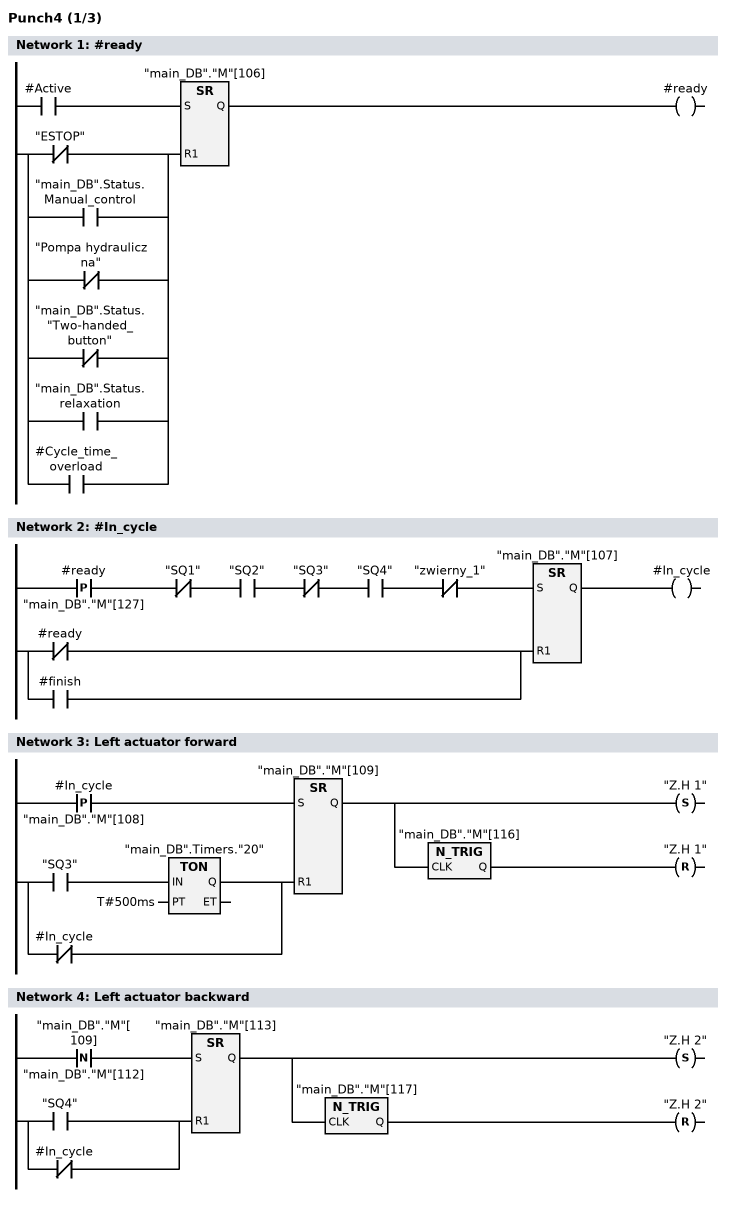
   RUNG wire#powerrail
      Contact( #Active )
      S_SR(operand := "main_DB"."M"[106], r1 := wire#w1)
      Coil( #ready )
   END_RUNG
   RUNG wire#powerrail
      I_Contact( "ESTOP" )
   END_RUNG wire#w1
   RUNG wire#powerrail
      Contact( "main_DB".Status.Manual_control )
   END_RUNG wire#w1
   RUNG wire#powerrail
      I_Contact( "Pompa hydrauliczna" )
   END_RUNG wire#w1
   RUNG wire#powerrail
      I_Contact( "main_DB".Status."Two-handed_button" )
   END_RUNG wire#w1
   RUNG wire#powerrail
      Contact( "main_DB".Status.relaxation )
   END_RUNG wire#w1
   RUNG wire#powerrail
      Contact( #Cycle_time_overload )
   END_RUNG wire#w1
   // the same network as SCL:
   IF #Active THEN
       "main_DB"."M"[106] := TRUE;   // SR flip-flop
   END_IF;
   IF NOT "ESTOP" OR "main_DB".Status.Manual_control OR NOT "Pompa hydrauliczna" OR NOT "main_DB".Status."Two-handed_button" OR "main_DB".Status.relaxation OR #Cycle_time_overload THEN
       "main_DB"."M"[106] := FALSE;
   END_IF;
   #ready := "main_DB"."M"[106];
END_REGION

REGION Network 2: #In_cycle
   RUNG wire#powerrail
      P_Contact(operand := #ready, bit := "main_DB"."M"[127])
      I_Contact( "SQ1" )
      Contact( "SQ2" )
      I_Contact( "SQ3" )
      Contact( "SQ4" )
      I_Contact( "zwierny_1" )
      S_SR(operand := "main_DB"."M"[107], r1 := wire#w1)
      Coil( #In_cycle )
   END_RUNG
   RUNG wire#powerrail
      I_Contact( #ready )
   END_RUNG wire#w1
   RUNG wire#powerrail
      Contact( #finish )
   END_RUNG wire#w1
   // the same network as SCL:
   #_w1 := #ready AND NOT "main_DB"."M"[127];   // rising edge of #ready
   "main_DB"."M"[127] := #ready;
   IF #_w1 AND NOT "SQ1" AND "SQ2" AND NOT "SQ3" AND "SQ4" AND NOT "zwierny_1" THEN
       "main_DB"."M"[107] := TRUE;   // SR flip-flop
   END_IF;
   IF NOT #ready OR #finish THEN "main_DB"."M"[107] := FALSE; END_IF;
   #In_cycle := "main_DB"."M"[107];
END_REGION

REGION Network 3: Left actuator forward
   #_w1 := #In_cycle AND NOT "main_DB"."M"[108];   // rising edge of #In_cycle
   "main_DB"."M"[108] := #In_cycle;
   "main_DB".Timers."20".TON(IN := "SQ3", PT := T#500ms);
   IF #_w1 THEN
       "main_DB"."M"[109] := TRUE;   // SR flip-flop
   END_IF;
   IF "main_DB".Timers."20".Q OR NOT #In_cycle THEN "main_DB"."M"[109] := FALSE; END_IF;
   IF "main_DB"."M"[109] THEN "Z.H 1" := TRUE; END_IF;
   #_w2 := "main_DB"."M"[109];
   #_w3 := NOT #_w2 AND "main_DB"."M"[116];   // falling edge
   "main_DB"."M"[116] := #_w2;
   IF #_w3 THEN "Z.H 1" := FALSE; END_IF;
END_REGION

REGION Network 4: Left actuator backward
   RUNG wire#powerrail
      N_Contact(operand := "main_DB"."M"[109], bit := "main_DB"."M"[112])
      S_SR(operand := "main_DB"."M"[113], r1 := wire#w1)
      wire#w2
      S_Coil( "Z.H 2" )
   END_RUNG
   RUNG wire#powerrail
      Contact( "SQ4" )
   END_RUNG wire#w1
   RUNG wire#powerrail
      I_Contact( #In_cycle )
   END_RUNG wire#w1
   RUNG wire#w2
      N_Trig( "main_DB"."M"[117] )
      R_Coil( "Z.H 2" )
   END_RUNG
   // the same network as SCL:
   #_w1 := NOT "main_DB"."M"[109] AND "main_DB"."M"[112];   // falling edge of "main_DB"."M"[109]
   "main_DB"."M"[112] := "main_DB"."M"[109];
   IF #_w1 THEN
       "main_DB"."M"[113] := TRUE;   // SR flip-flop
   END_IF;
   IF "SQ4" OR NOT #In_cycle THEN "main_DB"."M"[113] := FALSE; END_IF;
   IF "main_DB"."M"[113] THEN "Z.H 2" := TRUE; END_IF;
   #_w2 := "main_DB"."M"[113];
   #_w3 := NOT #_w2 AND "main_DB"."M"[117];   // falling edge
   "main_DB"."M"[117] := #_w2;
   IF #_w3 THEN "Z.H 2" := FALSE; END_IF;
END_REGION

REGION Network 5: Right actuator forward
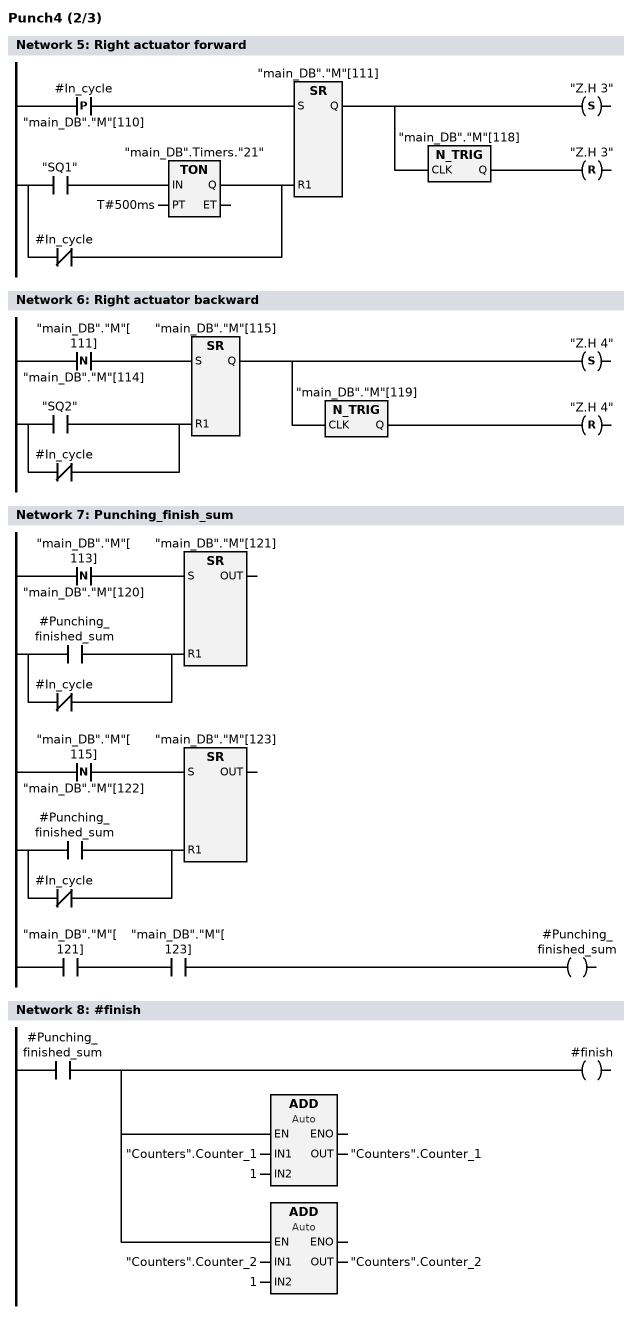
   #_w1 := #In_cycle AND NOT "main_DB"."M"[110];   // rising edge of #In_cycle
   "main_DB"."M"[110] := #In_cycle;
   "main_DB".Timers."21".TON(IN := "SQ1", PT := T#500ms);
   IF #_w1 THEN
       "main_DB"."M"[111] := TRUE;   // SR flip-flop
   END_IF;
   IF "main_DB".Timers."21".Q OR NOT #In_cycle THEN "main_DB"."M"[111] := FALSE; END_IF;
   IF "main_DB"."M"[111] THEN "Z.H 3" := TRUE; END_IF;
   #_w2 := "main_DB"."M"[111];
   #_w3 := NOT #_w2 AND "main_DB"."M"[118];   // falling edge
   "main_DB"."M"[118] := #_w2;
   IF #_w3 THEN "Z.H 3" := FALSE; END_IF;
END_REGION

REGION Network 6: Right actuator backward
   RUNG wire#powerrail
      N_Contact(operand := "main_DB"."M"[111], bit := "main_DB"."M"[114])
      S_SR(operand := "main_DB"."M"[115], r1 := wire#w1)
      wire#w2
      S_Coil( "Z.H 4" )
   END_RUNG
   RUNG wire#powerrail
      Contact( "SQ2" )
   END_RUNG wire#w1
   RUNG wire#powerrail
      I_Contact( #In_cycle )
   END_RUNG wire#w1
   RUNG wire#w2
      N_Trig( "main_DB"."M"[119] )
      R_Coil( "Z.H 4" )
   END_RUNG
   // the same network as SCL:
   #_w1 := NOT "main_DB"."M"[111] AND "main_DB"."M"[114];   // falling edge of "main_DB"."M"[111]
   "main_DB"."M"[114] := "main_DB"."M"[111];
   IF #_w1 THEN
       "main_DB"."M"[115] := TRUE;   // SR flip-flop
   END_IF;
   IF "SQ2" OR NOT #In_cycle THEN "main_DB"."M"[115] := FALSE; END_IF;
   IF "main_DB"."M"[115] THEN "Z.H 4" := TRUE; END_IF;
   #_w2 := "main_DB"."M"[115];
   #_w3 := NOT #_w2 AND "main_DB"."M"[119];   // falling edge
   "main_DB"."M"[119] := #_w2;
   IF #_w3 THEN "Z.H 4" := FALSE; END_IF;
END_REGION

REGION Network 7: Punching_finish_sum
   RUNG wire#powerrail
      N_Contact(operand := "main_DB"."M"[113], bit := "main_DB"."M"[120])
      S_SR(operand := "main_DB"."M"[121], r1 := wire#w1)
   END_RUNG
   RUNG wire#powerrail
      Contact( #Punching_finished_sum )
   END_RUNG wire#w1
   RUNG wire#powerrail
      I_Contact( #In_cycle )
   END_RUNG wire#w1
   RUNG wire#powerrail
      N_Contact(operand := "main_DB"."M"[115], bit := "main_DB"."M"[122])
      S_SR(operand := "main_DB"."M"[123], r1 := wire#w2)
   END_RUNG
   RUNG wire#powerrail
      Contact( #Punching_finished_sum )
   END_RUNG wire#w2
   RUNG wire#powerrail
      I_Contact( #In_cycle )
   END_RUNG wire#w2
   RUNG wire#powerrail
      Contact( "main_DB"."M"[121] )
      Contact( "main_DB"."M"[123] )
      Coil( #Punching_finished_sum )
   END_RUNG
   // the same network as SCL:
   #_w1 := NOT "main_DB"."M"[113] AND "main_DB"."M"[120];   // falling edge of "main_DB"."M"[113]
   "main_DB"."M"[120] := "main_DB"."M"[113];
   IF #_w1 THEN
       "main_DB"."M"[121] := TRUE;   // SR flip-flop
   END_IF;
   IF #Punching_finished_sum OR NOT #In_cycle THEN "main_DB"."M"[121] := FALSE; END_IF;
   #_w2 := NOT "main_DB"."M"[115] AND "main_DB"."M"[122];   // falling edge of "main_DB"."M"[115]
   "main_DB"."M"[122] := "main_DB"."M"[115];
   IF #_w2 THEN
       "main_DB"."M"[123] := TRUE;   // SR flip-flop
   END_IF;
   IF #Punching_finished_sum OR NOT #In_cycle THEN "main_DB"."M"[123] := FALSE; END_IF;
   #Punching_finished_sum := "main_DB"."M"[121] AND "main_DB"."M"[123];
END_REGION

REGION Network 8: #finish
   RUNG wire#powerrail
      Contact( #Punching_finished_sum )
      wire#w1
      Coil( #finish )
   END_RUNG
   RUNG wire#w1
      Add(in1 := "Counters".Counter_1, in2 := 1, out => "Counters".Counter_1)
   END_RUNG
   RUNG wire#w1
      Add(in1 := "Counters".Counter_2, in2 := 1, out => "Counters".Counter_2)
   END_RUNG
   // the same network as SCL:
   #finish := #Punching_finished_sum;
   IF #Punching_finished_sum THEN
       "Counters".Counter_1 := "Counters".Counter_1 + 1;
       "Counters".Counter_2 := "Counters".Counter_2 + 1;
   END_IF;
END_REGION

REGION Network 9: "Outputs_reset"
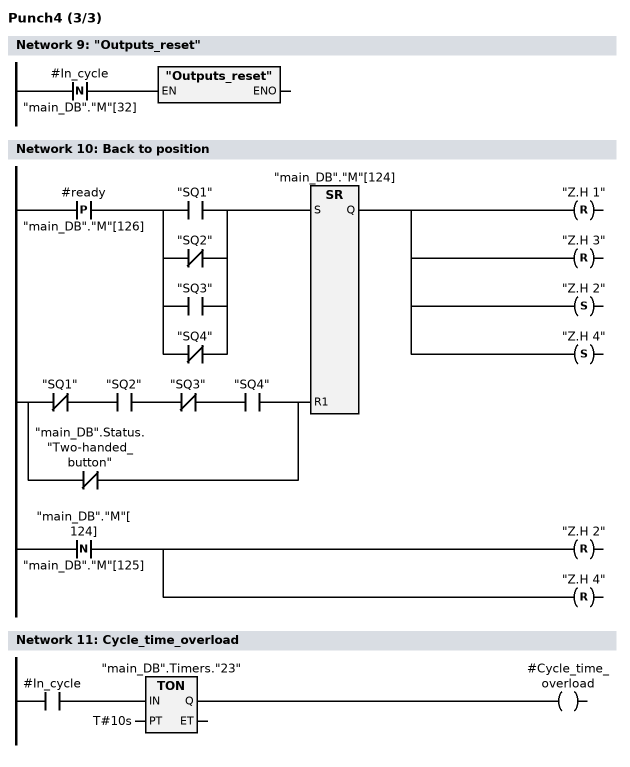
   RUNG wire#powerrail
      N_Contact(operand := #In_cycle, bit := "main_DB"."M"[32])
      "Outputs_reset"()
   END_RUNG
   // the same network as SCL:
   #_w1 := NOT #In_cycle AND "main_DB"."M"[32];   // falling edge of #In_cycle
   "main_DB"."M"[32] := #In_cycle;
   IF #_w1 THEN "Outputs_reset"(); END_IF;
END_REGION

REGION Network 10: Back to position
   RUNG wire#powerrail
      P_Contact(operand := #ready, bit := "main_DB"."M"[126])
      wire#w1
      Contact( "SQ1" )
      wire#w2
      S_SR(operand := "main_DB"."M"[124], r1 := wire#w3)
      wire#w4
      R_Coil( "Z.H 1" )
   END_RUNG
   RUNG wire#w1
      I_Contact( "SQ2" )
   END_RUNG wire#w2
   RUNG wire#w1
      Contact( "SQ3" )
   END_RUNG wire#w2
   RUNG wire#w1
      I_Contact( "SQ4" )
   END_RUNG wire#w2
   RUNG wire#powerrail
      I_Contact( "SQ1" )
      Contact( "SQ2" )
      I_Contact( "SQ3" )
      Contact( "SQ4" )
   END_RUNG wire#w3
   RUNG wire#powerrail
      I_Contact( "main_DB".Status."Two-handed_button" )
   END_RUNG wire#w3
   RUNG wire#w4
      R_Coil( "Z.H 3" )
   END_RUNG
   RUNG wire#w4
      S_Coil( "Z.H 2" )
   END_RUNG
   RUNG wire#w4
      S_Coil( "Z.H 4" )
   END_RUNG
   RUNG wire#powerrail
      N_Contact(operand := "main_DB"."M"[124], bit := "main_DB"."M"[125])
      wire#w5
      R_Coil( "Z.H 2" )
   END_RUNG
   RUNG wire#w5
      R_Coil( "Z.H 4" )
   END_RUNG
   // the same network as SCL:
   #_w1 := #ready AND NOT "main_DB"."M"[126];   // rising edge of #ready
   "main_DB"."M"[126] := #ready;
   IF #_w1 AND ("SQ1" OR NOT "SQ2" OR "SQ3" OR NOT "SQ4") THEN
       "main_DB"."M"[124] := TRUE;   // SR flip-flop
   END_IF;
   IF (NOT "SQ1" AND "SQ2" AND NOT "SQ3" AND "SQ4") OR NOT "main_DB".Status."Two-handed_button" THEN
       "main_DB"."M"[124] := FALSE;
   END_IF;
   IF "main_DB"."M"[124] THEN
       "Z.H 1" := FALSE;
       "Z.H 3" := FALSE;
       "Z.H 2" := TRUE;
       "Z.H 4" := TRUE;
   END_IF;
   #_w2 := NOT "main_DB"."M"[124] AND "main_DB"."M"[125];   // falling edge of "main_DB"."M"[124]
   "main_DB"."M"[125] := "main_DB"."M"[124];
   IF #_w2 THEN
       "Z.H 2" := FALSE;
       "Z.H 4" := FALSE;
   END_IF;
END_REGION

REGION Network 11: Cycle_time_overload
   "main_DB".Timers."23".TON(IN := #In_cycle, PT := T#10s);
   #Cycle_time_overload := "main_DB".Timers."23".Q;
END_REGION
END_FUNCTION_BLOCK

FUNCTION_BLOCK "Punch5"   // FB6, LAD
{ S7_Optimized_Access := 'TRUE' }
VERSION : 0.1
   VAR_INPUT
      Active : Bool;
   END_VAR
   VAR
      finish : Bool;
      Cycle_time_overload : Bool;
   END_VAR
   VAR_TEMP
      In_cycle : Bool;
      ready : Bool;
   END_VAR
   VAR_TEMP   // added for the SCL form of the ladder/FBD networks
      _w1 : Bool;
      _w2 : Bool;
      _w3 : Bool;
   END_VAR
BEGIN

REGION Network 1: #ready
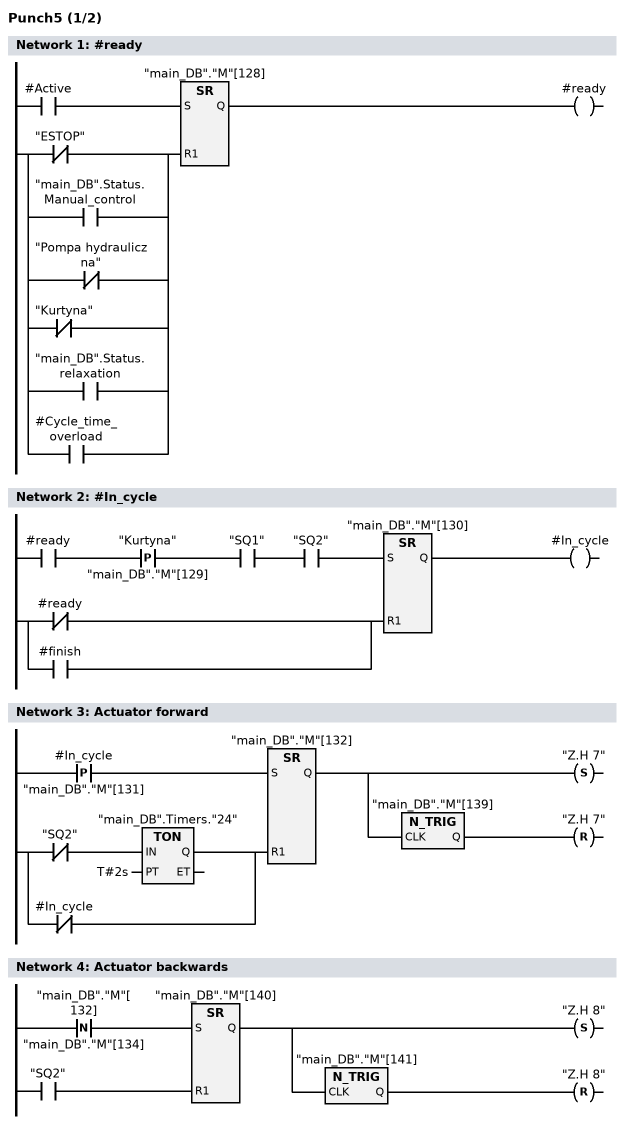
   RUNG wire#powerrail
      Contact( #Active )
      S_SR(operand := "main_DB"."M"[128], r1 := wire#w1)
      Coil( #ready )
   END_RUNG
   RUNG wire#powerrail
      I_Contact( "ESTOP" )
   END_RUNG wire#w1
   RUNG wire#powerrail
      Contact( "main_DB".Status.Manual_control )
   END_RUNG wire#w1
   RUNG wire#powerrail
      I_Contact( "Pompa hydrauliczna" )
   END_RUNG wire#w1
   RUNG wire#powerrail
      I_Contact( "Kurtyna" )
   END_RUNG wire#w1
   RUNG wire#powerrail
      Contact( "main_DB".Status.relaxation )
   END_RUNG wire#w1
   RUNG wire#powerrail
      Contact( #Cycle_time_overload )
   END_RUNG wire#w1
   // the same network as SCL:
   IF #Active THEN
       "main_DB"."M"[128] := TRUE;   // SR flip-flop
   END_IF;
   IF NOT "ESTOP" OR "main_DB".Status.Manual_control OR NOT "Pompa hydrauliczna" OR NOT "Kurtyna" OR "main_DB".Status.relaxation OR #Cycle_time_overload THEN
       "main_DB"."M"[128] := FALSE;
   END_IF;
   #ready := "main_DB"."M"[128];
END_REGION

REGION Network 2: #In_cycle
   RUNG wire#powerrail
      Contact( #ready )
      P_Contact(operand := "Kurtyna", bit := "main_DB"."M"[129])
      Contact( "SQ1" )
      Contact( "SQ2" )
      S_SR(operand := "main_DB"."M"[130], r1 := wire#w1)
      Coil( #In_cycle )
   END_RUNG
   RUNG wire#powerrail
      I_Contact( #ready )
   END_RUNG wire#w1
   RUNG wire#powerrail
      Contact( #finish )
   END_RUNG wire#w1
   // the same network as SCL:
   #_w1 := #ready AND "Kurtyna" AND NOT "main_DB"."M"[129];   // rising edge of "Kurtyna"
   "main_DB"."M"[129] := "Kurtyna";
   IF #_w1 AND "SQ1" AND "SQ2" THEN
       "main_DB"."M"[130] := TRUE;   // SR flip-flop
   END_IF;
   IF NOT #ready OR #finish THEN "main_DB"."M"[130] := FALSE; END_IF;
   #In_cycle := "main_DB"."M"[130];
END_REGION

REGION Network 3: Actuator forward
   #_w1 := #In_cycle AND NOT "main_DB"."M"[131];   // rising edge of #In_cycle
   "main_DB"."M"[131] := #In_cycle;
   "main_DB".Timers."24".TON(IN := NOT "SQ2", PT := T#2s);
   IF #_w1 THEN
       "main_DB"."M"[132] := TRUE;   // SR flip-flop
   END_IF;
   IF "main_DB".Timers."24".Q OR NOT #In_cycle THEN "main_DB"."M"[132] := FALSE; END_IF;
   IF "main_DB"."M"[132] THEN "Z.H 7" := TRUE; END_IF;
   #_w2 := "main_DB"."M"[132];
   #_w3 := NOT #_w2 AND "main_DB"."M"[139];   // falling edge
   "main_DB"."M"[139] := #_w2;
   IF #_w3 THEN "Z.H 7" := FALSE; END_IF;
END_REGION

REGION Network 4: Actuator backwards
   RUNG wire#powerrail
      N_Contact(operand := "main_DB"."M"[132], bit := "main_DB"."M"[134])
      S_SR(operand := "main_DB"."M"[140], r1 := wire#w1)
      wire#w2
      S_Coil( "Z.H 8" )
   END_RUNG
   RUNG wire#powerrail
      Contact( "SQ2" )
   END_RUNG wire#w1
   RUNG wire#w2
      N_Trig( "main_DB"."M"[141] )
      R_Coil( "Z.H 8" )
   END_RUNG
   // the same network as SCL:
   #_w1 := NOT "main_DB"."M"[132] AND "main_DB"."M"[134];   // falling edge of "main_DB"."M"[132]
   "main_DB"."M"[134] := "main_DB"."M"[132];
   IF #_w1 THEN
       "main_DB"."M"[140] := TRUE;   // SR flip-flop
   END_IF;
   IF "SQ2" THEN "main_DB"."M"[140] := FALSE; END_IF;
   IF "main_DB"."M"[140] THEN "Z.H 8" := TRUE; END_IF;
   #_w2 := "main_DB"."M"[140];
   #_w3 := NOT #_w2 AND "main_DB"."M"[141];   // falling edge
   "main_DB"."M"[141] := #_w2;
   IF #_w3 THEN "Z.H 8" := FALSE; END_IF;
END_REGION

REGION Network 5: #finish
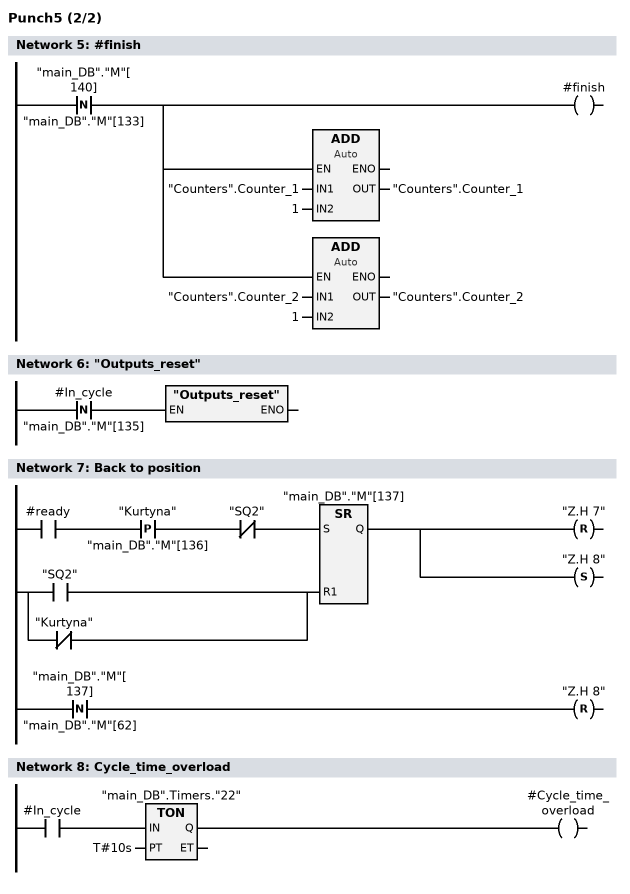
   RUNG wire#powerrail
      N_Contact(operand := "main_DB"."M"[140], bit := "main_DB"."M"[133])
      wire#w1
      Coil( #finish )
   END_RUNG
   RUNG wire#w1
      Add(in1 := "Counters".Counter_1, in2 := 1, out => "Counters".Counter_1)
   END_RUNG
   RUNG wire#w1
      Add(in1 := "Counters".Counter_2, in2 := 1, out => "Counters".Counter_2)
   END_RUNG
   // the same network as SCL:
   #_w1 := NOT "main_DB"."M"[140] AND "main_DB"."M"[133];   // falling edge of "main_DB"."M"[140]
   "main_DB"."M"[133] := "main_DB"."M"[140];
   #finish := #_w1;
   IF #_w1 THEN
       "Counters".Counter_1 := "Counters".Counter_1 + 1;
       "Counters".Counter_2 := "Counters".Counter_2 + 1;
   END_IF;
END_REGION

REGION Network 6: "Outputs_reset"
   RUNG wire#powerrail
      N_Contact(operand := #In_cycle, bit := "main_DB"."M"[135])
      "Outputs_reset"()
   END_RUNG
   // the same network as SCL:
   #_w1 := NOT #In_cycle AND "main_DB"."M"[135];   // falling edge of #In_cycle
   "main_DB"."M"[135] := #In_cycle;
   IF #_w1 THEN "Outputs_reset"(); END_IF;
END_REGION

REGION Network 7: Back to position
   RUNG wire#powerrail
      Contact( #ready )
      P_Contact(operand := "Kurtyna", bit := "main_DB"."M"[136])
      I_Contact( "SQ2" )
      S_SR(operand := "main_DB"."M"[137], r1 := wire#w1)
      wire#w2
      R_Coil( "Z.H 7" )
   END_RUNG
   RUNG wire#powerrail
      Contact( "SQ2" )
   END_RUNG wire#w1
   RUNG wire#powerrail
      I_Contact( "Kurtyna" )
   END_RUNG wire#w1
   RUNG wire#w2
      S_Coil( "Z.H 8" )
   END_RUNG
   RUNG wire#powerrail
      N_Contact(operand := "main_DB"."M"[137], bit := "main_DB"."M"[62])
      R_Coil( "Z.H 8" )
   END_RUNG
   // the same network as SCL:
   #_w1 := #ready AND "Kurtyna" AND NOT "main_DB"."M"[136];   // rising edge of "Kurtyna"
   "main_DB"."M"[136] := "Kurtyna";
   IF #_w1 AND NOT "SQ2" THEN
       "main_DB"."M"[137] := TRUE;   // SR flip-flop
   END_IF;
   IF "SQ2" OR NOT "Kurtyna" THEN "main_DB"."M"[137] := FALSE; END_IF;
   IF "main_DB"."M"[137] THEN
       "Z.H 7" := FALSE;
       "Z.H 8" := TRUE;
   END_IF;
   #_w2 := NOT "main_DB"."M"[137] AND "main_DB"."M"[62];   // falling edge of "main_DB"."M"[137]
   "main_DB"."M"[62] := "main_DB"."M"[137];
   IF #_w2 THEN "Z.H 8" := FALSE; END_IF;
END_REGION

REGION Network 8: Cycle_time_overload
   "main_DB".Timers."22".TON(IN := #In_cycle, PT := T#10s);
   #Cycle_time_overload := "main_DB".Timers."22".Q;
END_REGION
END_FUNCTION_BLOCK

(* ===== HMI "HMI_RT_1" =====
system functions are stored by id; their names below are inferred from use
connection "HMI_Connection_2": ETHERNET, SMART_S7_1200_OMS

HMI tags "Default tag table"
   "Screen_number" : Int, internal
   "main_DB_Button_Screen_1_Z.P 0" : Bool = PLC main_DB.Button.Screen_2."Z.P 0", 100 ms
   "main_DB_Button_Screen_1_Z.P 1" : Bool = PLC main_DB.Button.Screen_2."Z.P 1", 100 ms
   "main_DB_Button_Screen_1_Z.P 3" : Bool = PLC main_DB.Button.Screen_2."Z.P 3", 100 ms
   "main_DB_Button_Screen_1_Z.P 2" : Bool = PLC main_DB.Button.Screen_2."Z.P 2", 100 ms
   "main_DB_Button_Screen_1_Z.P 4" : Bool = PLC main_DB.Button.Screen_2."Z.P 4", 100 ms
   "main_DB_Button_Screen_1_Z.H 1" : Bool = PLC main_DB.Button.Screen_2."Z.H 1", 100 ms
   "main_DB_Button_Screen_1_Z.H 2" : Bool = PLC main_DB.Button.Screen_2."Z.H 2", 100 ms
   "main_DB_Button_Screen_1_Z.H 3" : Bool = PLC main_DB.Button.Screen_2."Z.H 3", 100 ms
   "main_DB_Button_Screen_1_Z.H 4" : Bool = PLC main_DB.Button.Screen_2."Z.H 4", 100 ms
   "main_DB_Button_Screen_1_Z.H 5" : Bool = PLC main_DB.Button.Screen_2."Z.H 5", 100 ms
   "main_DB_Button_Screen_1_Z.H 6" : Bool = PLC main_DB.Button.Screen_2."Z.H 6", 100 ms
   "main_DB_Button_Screen_1_Z.H 7" : Bool = PLC main_DB.Button.Screen_2."Z.H 7", 100 ms
   "main_DB_Button_Screen_1_Z.H 8" : Bool = PLC main_DB.Button.Screen_2."Z.H 8", 100 ms
   "main_DB_Button_Screen_1_Z.H 0" : Bool = PLC main_DB.Button.Screen_2."Z.H 0", 100 ms
   "Z.P 0" : Bool = PLC "Z.P 0" AT %Q12.0, 100 ms
   "Z.P 1" : Bool = PLC "Z.P 1" AT %Q12.1, 100 ms
   "Z.P 2" : Bool = PLC "Z.P 2" AT %Q12.2, 100 ms
   "Z.P 3" : Bool = PLC "Z.P 3" AT %Q12.3, 100 ms
   "Z.P 4" : Bool = PLC "Z.P 4" AT %Q12.4, 100 ms
   "Z.H 1" : Bool = PLC "Z.H 1" AT %Q0.1, 100 ms
   "Z.H 2" : Bool = PLC "Z.H 2" AT %Q0.2, 100 ms
   "Z.H 3" : Bool = PLC "Z.H 3" AT %Q0.3, 100 ms
   "Z.H 4" : Bool = PLC "Z.H 4" AT %Q0.4, 100 ms
   "Z.H 5" : Bool = PLC "Z.H 5" AT %Q0.5, 100 ms
   "Z.H 6" : Bool = PLC "Z.H 6" AT %Q0.6, 100 ms
   "Z.H 7" : Bool = PLC "Z.H 7" AT %Q0.7, 100 ms
   "Z.H 8" : Bool = PLC "Z.H 8" AT %Q1.0, 100 ms
   "Z.H 0" : Bool = PLC "Z.H 0" AT %Q0.0, 100 ms
   "main_DB_Button_Screen_0_Reset_counter_1" : Bool = PLC main_DB.Button.Screen_0.Reset_counter_1, 100 ms
   "main_DB_Button_Screen_0_Reset_counter_2" : Bool = PLC main_DB.Button.Screen_0.Reset_counter_2, 100 ms
   "main_DB_Status_Browsing_punch" : Bool = PLC main_DB.Status.Browsing_punch, 100 ms
   "Counters_Counter_1" : Int = PLC Counters.Counter_1, 500 ms
   "Counters_Counter_2" : Int = PLC Counters.Counter_2, 500 ms
   "main_DB_Status_Manual_control" : Bool = PLC main_DB.Status.Manual_control, 100 ms
   "main_DB_Button_Screen_1_Manual_control" : Bool = PLC main_DB.Button.Screen_2.Manual_control, 100 ms
   "main_DB_Button_Screen_1_Hydraulic_Pump" : Bool = PLC main_DB.Button.Screen_2.Hydraulic_Pump, 100 ms
   "Pompa hydrauliczna" : Bool = PLC "Pompa hydrauliczna" AT %Q13.4, 100 ms
   "main_DB_var_Result_punch" : Byte = PLC main_DB.var.Result_punch, 100 ms
   "main_DB_var_Connected_punch" : Byte = PLC main_DB.var.Connected_punch, 100 ms
   "main_DB_Button_Template_Browsed_punch_-" : Bool = PLC main_DB.Button.Template.Browsed_punch_-, 100 ms
   "main_DB_Button_Template_Browsed_punch_+" : Bool = PLC main_DB.Button.Template.Browsed_punch_+, 100 ms
   "main_DB_var_Hydraulic_oil_pressure" : Real = PLC main_DB.var.Hydraulic_oil_pressure, 100 ms
   "main_DB_var_Descryption Z.P 1" : String[254] = PLC main_DB.var."Descryption Z.P 1", 500 ms
   "main_DB_var_Descryption Z.P 2" : String[254] = PLC main_DB.var."Descryption Z.P 2", 500 ms
   "main_DB_var_Descryption Z.P 3" : String[254] = PLC main_DB.var."Descryption Z.P 3", 500 ms
   "main_DB_var_Descryption Z.P 4" : String[254] = PLC main_DB.var."Descryption Z.P 4", 500 ms
   "main_DB_var_Descryption Z.H 1" : String[254] = PLC main_DB.var."Descryption Z.H 1", 500 ms
   "main_DB_var_Descryption Z.H 2" : String[254] = PLC main_DB.var."Descryption Z.H 2", 500 ms
   "main_DB_var_Descryption Z.H 3" : String[254] = PLC main_DB.var."Descryption Z.H 3", 500 ms
   "main_DB_var_Descryption Z.H 4" : String[254] = PLC main_DB.var."Descryption Z.H 4", 500 ms
   "main_DB_var_Descryption Z.H 5" : String[254] = PLC main_DB.var."Descryption Z.H 5", 500 ms
   "main_DB_var_Descryption Z.H 6" : String[254] = PLC main_DB.var."Descryption Z.H 6", 500 ms
   "main_DB_var_Descryption Z.H 7" : String[254] = PLC main_DB.var."Descryption Z.H 7", 500 ms
   "main_DB_var_Descryption Z.H 8" : String[254] = PLC main_DB.var."Descryption Z.H 8", 500 ms
   "SQ1" : Bool = PLC SQ1 AT %I1.0, 100 ms
   "SQ2" : Bool = PLC SQ2 AT %I1.1, 100 ms
   "SQ3" : Bool = PLC SQ3 AT %I1.2, 100 ms
   "SQ4" : Bool = PLC SQ4 AT %I1.3, 100 ms
   "SQ5" : Bool = PLC SQ5 AT %I1.4, 100 ms
   "SQ6" : Bool = PLC SQ6 AT %I1.5, 100 ms
   "zwierny_1" : Bool = PLC zwierny_1 AT %I8.6, 100 ms
   "zwierny_2" : Bool = PLC zwierny_2 AT %I8.7, 100 ms
   "zwierny_3" : Bool = PLC zwierny_3 AT %I9.0, 100 ms
   "zwierny_4" : Bool = PLC zwierny_4 AT %I9.1, 100 ms
   "zwierny_5" : Bool = PLC zwierny_5 AT %I9.2, 100 ms
   "zwierny_6" : Bool = PLC zwierny_6 AT %I9.3, 100 ms
   "main_DB_var_Descryption SQ 1" : String[254] = PLC main_DB.var."Descryption SQ 1", 500 ms
   "main_DB_var_Descryption SQ 2" : String[254] = PLC main_DB.var."Descryption SQ 2", 500 ms
   "main_DB_var_Descryption SQ 3" : String[254] = PLC main_DB.var."Descryption SQ 3", 500 ms
   "main_DB_var_Descryption SQ 4" : String[254] = PLC main_DB.var."Descryption SQ 4", 500 ms
   "main_DB_var_Descryption SQ 5" : String[254] = PLC main_DB.var."Descryption SQ 5", 500 ms
   "main_DB_var_Descryption SQ 6" : String[254] = PLC main_DB.var."Descryption SQ 6", 500 ms
   "main_DB_var_Descryption contact_sensor 1" : String[254] = PLC main_DB.var."Descryption contact_sensor 1", 500 ms
   "main_DB_var_Descryption contact_sensor 2" : String[254] = PLC main_DB.var."Descryption contact_sensor 2", 500 ms
   "main_DB_var_Descryption contact_sensor 3" : String[254] = PLC main_DB.var."Descryption contact_sensor 3", 500 ms
   "main_DB_var_Descryption contact_sensor 4" : String[254] = PLC main_DB.var."Descryption contact_sensor 4", 500 ms
   "main_DB_var_Descryption contact_sensor 5" : String[254] = PLC main_DB.var."Descryption contact_sensor 5", 500 ms
   "main_DB_var_Descryption contact_sensor 6" : String[254] = PLC main_DB.var."Descryption contact_sensor 6", 500 ms
   "czujnik ciśnienia powietrza" : Bool = PLC "czujnik ciśnienia powietrza" AT %I0.0, 100 ms
   "main_DB_Status_relaxation" : Bool = PLC main_DB.Status.relaxation, 100 ms
   "main_DB_Button_Screen_2_Relaxation" : Bool = PLC main_DB.Button.Screen_2.Relaxation, 100 ms
   "main_DB_var_Lubrication_frequency" : Int = PLC main_DB.var.Lubrication_frequency, 500 ms
   "main_DB_var_Lubrication_dur" : Time = PLC main_DB.var.Lubrication_dur, 500 ms
   "main_DB_Button_Screen_0_Lubrication_test_1" : Bool = PLC main_DB.Button.Screen_0.Lubrication_test_1, 100 ms
   "main_DB_Button_Screen_0_Lubrication_test_2" : Bool = PLC main_DB.Button.Screen_0.Lubrication_test_2, 100 ms

Template "KTP700 logo & menu" 800x480
   GraphicView "Template_Graphic view_1" at 8,6 size 400x68; Picture "INNOWACJA"
   Button "Button_1" at 720,30 size 64x64; TextOff '0'
      Appearance <- "Screen_number"
      on Press: ActivateScreen("Screen_0", 0)
   Button "Button_2" at 720,386 size 64x64; TextOff '3'
      Appearance <- "Screen_number"
      on Press: ActivateScreen("Screen_3", 0)
   Button "Button_3" at 720,148 size 64x64; TextOff '1'
      Appearance <- "Screen_number"
      on Press: ActivateScreen("Screen_1", 0)
   Button "Button_4" at 720,267 size 64x64; TextOff '2'
      Appearance <- "Screen_number"
      on Press: ActivateScreen("Screen_2", 0)
   IOField "I/O field_1" at 539,12 size 54x54; FormatPattern 99
      ProcessValue <- "main_DB_var_Result_punch"
   Button "Button_5" at 613,12 size 54x54; TextOff 'Reset'; PictureOff "Graphic_2"
      on Press: function_b14e0dd5("main_DB_Button_Template_Browsed_punch_+", 0)
      Visibility <- "main_DB_var_Connected_punch"
   Button "Button_6" at 469,12 size 54x54; TextOff 'Reset'; PictureOff "Graphic_3"
      on Press: function_b14e0dd5("main_DB_Button_Template_Browsed_punch_-", 0)
      Visibility <- "main_DB_var_Connected_punch"

screen "Screen_0" 800x480, template "KTP700 logo & menu"
   on GenerateScreen: SetTag("Screen_number", 0)
   IOField "I/O field_2" at 14,413 size 140x54; FormatPattern 9999999
      ProcessValue <- "Counters_Counter_2"
   TextField "Text field_2" at 14,381 size 209x32; Text 'Licznik zmianowy'
   IOField "I/O field_3" at 14,325 size 140x54; FormatPattern 9999999
      ProcessValue <- "Counters_Counter_1"
   TextField "Text field_3" at 14,290 size 155x32; Text 'Licznik sztuk'
   Button "Button_1" at 190,325 size 54x54; TextOff 'Reset'
      on Press: function_b14e0dd5("main_DB_Button_Screen_0_Reset_counter_1", 0)
      Appearance <- "main_DB_Button_Screen_0_Reset_counter_1"
   Button "Button_2" at 190,413 size 54x54; TextOff 'Reset'
      on Press: function_b14e0dd5("main_DB_Button_Screen_0_Reset_counter_2", 0)
      Appearance <- "main_DB_Button_Screen_0_Reset_counter_2"
   Button "Button_7" at 382,122 size 55x55; TextOff '1'
      Appearance <- "zwierny_1"
   Button "Button_8" at 382,179 size 55x55; TextOff '2'
      Appearance <- "zwierny_2"
   Button "Button_9" at 382,237 size 55x55; TextOff '3'
      Appearance <- "zwierny_3"
   Button "Button_10" at 382,295 size 55x55; TextOff '4'
      Appearance <- "zwierny_4"
   Button "Button_11" at 382,353 size 55x55; TextOff '5'
      Appearance <- "zwierny_5"
   Button "Button_12" at 382,411 size 55x55; TextOff '6'
      Appearance <- "zwierny_6"
   IOField "I/O field_7" at 441,134 size 275x32; FormatPattern ????????????????????????????????????????????????????????????????????????????????
      ProcessValue <- "main_DB_var_Descryption contact_sensor 1"
   IOField "I/O field_8" at 441,191 size 275x32; FormatPattern ????????????????????????????????????????????????????????????????????????????????
      ProcessValue <- "main_DB_var_Descryption contact_sensor 2"
   IOField "I/O field_9" at 441,249 size 275x32; FormatPattern ????????????????????????????????????????????????????????????????????????????????
      ProcessValue <- "main_DB_var_Descryption contact_sensor 3"
   IOField "I/O field_10" at 441,307 size 275x32; FormatPattern ????????????????????????????????????????????????????????????????????????????????
      ProcessValue <- "main_DB_var_Descryption contact_sensor 4"
   IOField "I/O field_11" at 441,365 size 275x32; FormatPattern ????????????????????????????????????????????????????????????????????????????????
      ProcessValue <- "main_DB_var_Descryption contact_sensor 5"
   IOField "I/O field_12" at 441,423 size 275x32; FormatPattern ????????????????????????????????????????????????????????????????????????????????
      ProcessValue <- "main_DB_var_Descryption contact_sensor 6"
   TextField "Text field_1" at 358,85 size 367x34; Text 'Kołki stykowe'
   IOField "I/O field_1" at 14,236 size 140x54; FormatPattern s9999999999
      ProcessValue <- "main_DB_var_Lubrication_dur"
   TextField "Text field_4" at 14,204 size 268x32; Text 'Czas smarowania [ms]'
   IOField "I/O field_4" at 14,148 size 140x54; FormatPattern 9999999
      ProcessValue <- "main_DB_var_Lubrication_frequency"
   TextField "Text field_5" at 14,88 size 255x60; Text 'Częstość smarowania [l. cykli] (1-4)'
   Button "Button_3" at 244,236 size 54x54; TextOff 'Test 2'
      on Press: function_b14e0dd5("main_DB_Button_Screen_0_Lubrication_test_2", 0)
      Appearance <- "main_DB_Button_Screen_0_Reset_counter_1"
   Button "Button_4" at 190,236 size 54x54; TextOff 'Test 1'
      on Press: function_b14e0dd5("main_DB_Button_Screen_0_Lubrication_test_1", 0)
      Appearance <- "main_DB_Button_Screen_0_Reset_counter_2"

screen "Screen_1" 800x480, template "KTP700 logo & menu"
   on GenerateScreen: SetTag("Screen_number", 1)
   GraphicView "1" at 46,82 size 631x398; Picture "40214 - rysunek_4"
      Visibility <- "main_DB_var_Result_punch"
   TextField "Text field_1" at 278,260 size 215x43; Text 'Brak rysunku'

